LIN {X 0,Y 258.679,Z 819.95,A -85,B 0,C 180,E1 17212.36,E2 17212.36} C_VEL
LIN {X 0,Y 264.496,Z 801.8,A -85,B 0,C 180,E1 17220.057,E2 17220.057} C_VEL
LIN {X 0,Y 273.241,Z 778.314,A -85,B 0,C 180,E1 17227.008,E2 17227.008} C_VEL
LIN {X 0,Y 284.7,Z 748.46,A -85,B 0,C 180,E1 17233.215,E2 17233.215} C_VEL
LIN {X 0,Y 297.106,Z 713.594,A -85,B 0,C 180,E1 17238.218,E2 17238.218} C_VEL
LIN {X 0,Y 308.167,Z 677.358,A -85,B 0,C 180,E1 17241.821,E2 17241.821} C_VEL
LIN {X 0,Y 310.723,Z 665.135,A -85,B 0,C 180,E1 17242.87,E2 17242.87} C_VEL
LIN {X 0,Y 299.112,Z 634.221,A -85,B 0,C 180,E1 17248.073,E2 17248.073} C_VEL
LIN {X 0,Y 298.499,Z 632.776,A -85,B 0,C 180,E1 17248.333,E2 17248.333} C_VEL
LIN {X 0,Y 292.941,Z 625.387,A -85,B 0,C 180,E1 17250.142,E2 17250.142} C_VEL
LIN {X 0,Y 282.487,Z 614.328,A -85,B 0,C 180,E1 17253.334,E2 17253.334} C_VEL
LIN {X 0,Y 266.688,Z 585.354,A -85,B 0,C 180,E1 17259.767,E2 17259.767} C_VEL
LIN {X 0,Y 252.053,Z 561.723,A -85,B 0,C 180,E1 17266.216,E2 17266.216} C_VEL
LIN {X 0,Y 248.005,Z 555.389,A -85,B 0,C 180,E1 17268.238,E2 17268.238} C_VEL
LIN {X 0,Y 245.574,Z 550.181,A -85,B 0,C 180,E1 17269.651,E2 17269.651} C_VEL
LIN {X 0,Y 246.167,Z 549.53,A -85,B 0,C 180,E1 17276.481,E2 17276.481} C_VEL
LIN {X 0,Y 246.53,Z 549.53,A -85,B 0,C 180,E1 17280.007,E2 17280.007} C_VEL
LIN {X 0,Y 245.808,Z 549.53,A -85,B 0,C 180,E1 17287.084,E2 17287.084} C_VEL
LIN {X 0,Y 245.168,Z 549.53,A -85,B 0,C 180,E1 17294.309,E2 17294.309} C_VEL
LIN {X 0,Y 244.572,Z 549.53,A -85,B 0,C 180,E1 17301.812,E2 17301.812} C_VEL
LIN {X 0,Y 244.107,Z 549.53,A -85,B 0,C 180,E1 17309.756,E2 17309.756} C_VEL
LIN {X 0,Y 243.773,Z 549.53,A -85,B 0,C 180,E1 17318.404,E2 17318.404} C_VEL
LIN {X 0,Y 243.66,Z 549.53,A -85,B 0,C 180,E1 17326.882,E2 17326.882} C_VEL
LIN {X 0,Y 243.817,Z 549.53,A -85,B 0,C 180,E1 17336.023,E2 17336.023} C_VEL
LIN {X 0,Y 244.37,Z 549.53,A -85,B 0,C 180,E1 17344.299,E2 17344.299} C_VEL
LIN {X 0,Y 244.862,Z 549.53,A -85,B 0,C 180,E1 17351.993,E2 17351.993} C_VEL
LIN {X 0,Y 245.584,Z 549.53,A -85,B 0,C 180,E1 17360.585,E2 17360.585} C_VEL
LIN {X 0,Y 246.312,Z 549.696,A -85,B 0,C 180,E1 17368.13,E2 17368.13} C_VEL
LIN {X 0,Y 248.757,Z 555.053,A -85,B 0,C 180,E1 17369.566,E2 17369.566} C_VEL
LIN {X 0,Y 251.1,Z 558.751,A -85,B 0,C 180,E1 17370.757,E2 17370.757} C_VEL
LIN {X 0,Y 263.419,Z 580.328,A -85,B 0,C 180,E1 17376.986,E2 17376.986} C_VEL
LIN {X 0,Y 276.368,Z 608.507,A -85,B 0,C 180,E1 17383.801,E2 17383.801} C_VEL
LIN {X 0,Y 286.352,Z 636.818,A -85,B 0,C 180,E1 17389.901,E2 17389.901} C_VEL
LIN {X 0,Y 293.204,Z 665.582,A -85,B 0,C 180,E1 17395.869,E2 17395.869} C_VEL
LIN {X 0,Y 292.815,Z 670.961,A -85,B 0,C 180,E1 17396.759,E2 17396.759} C_VEL
LIN {X 0,Y 280.786,Z 703.835,A -85,B 0,C 180,E1 17401.766,E2 17401.766} C_VEL
LIN {X 0,Y 269.635,Z 731.204,A -85,B 0,C 180,E1 17407.633,E2 17407.633} C_VEL
LIN {X 0,Y 260.58,Z 753.078,A -85,B 0,C 180,E1 17414.208,E2 17414.208} C_VEL
LIN {X 0,Y 253.504,Z 771.169,A -85,B 0,C 180,E1 17421.942,E2 17421.942} C_VEL
LIN {X 0,Y 249.653,Z 783.095,A -85,B 0,C 180,E1 17429.414,E2 17429.414} C_VEL
LIN {X 0,Y 247.652,Z 790.352,A -85,B 0,C 180,E1 17436.502,E2 17436.502} C_VEL
LIN {X 0,Y 246.858,Z 793.707,A -85,B 0,C 180,E1 17442.134,E2 17442.134} C_VEL
LIN {X 0,Y 247.311,Z 795.056,A -85,B 0,C 180,E1 17449.41,E2 17449.41} C_VEL
LIN {X 0,Y 249.686,Z 792.262,A -85,B 0,C 180,E1 17458.054,E2 17458.054} C_VEL
LIN {X 0,Y 255.266,Z 783.653,A -85,B 0,C 180,E1 17467.662,E2 17467.662} C_VEL
LIN {X 0,Y 265.509,Z 769.339,A -85,B 0,C 180,E1 17476.559,E2 17476.559} C_VEL
LIN {X 0,Y 280.933,Z 748.975,A -85,B 0,C 180,E1 17484.68,E2 17484.68} C_VEL
LIN {X 0,Y 304.019,Z 719.389,A -85,B 0,C 180,E1 17492.361,E2 17492.361} C_VEL
LIN {X 0,Y 315.827,Z 704.851,A -85,B 0,C 180,E1 17495.111,E2 17495.111} C_VEL
LIN {X 0,Y 317.542,Z 702.998,A -85,B 0,C 180,E1 17495.846,E2 17495.846} C_VEL
LIN {X 0,Y 291.865,Z 741.185,A -85,B 0,C 180,E1 17501.778,E2 17501.778} C_VEL
LIN {X 0,Y 271.633,Z 776.074,A -85,B 0,C 180,E1 17509.609,E2 17509.609} C_VEL
LIN {X 0,Y 258.491,Z 802.354,A -85,B 0,C 180,E1 17518.185,E2 17518.185} C_VEL
LIN {X 0,Y 251.091,Z 820.776,A -85,B 0,C 180,E1 17526.923,E2 17526.923} C_VEL
LIN {X 0,Y 247.867,Z 833.059,A -85,B 0,C 180,E1 17535.856,E2 17535.856} C_VEL
LIN {X 0,Y 247.295,Z 838.614,A -85,B 0,C 180,E1 17542.965,E2 17542.965} C_VEL
LIN {X 0,Y 247.721,Z 840.447,A -85,B 0,C 180,E1 17549.998,E2 17549.998} C_VEL
LIN {X 0,Y 247.391,Z 838.37,A -85,B 0,C 180,E1 17557.029,E2 17557.029} C_VEL
LIN {X 0,Y 248.174,Z 831.193,A -85,B 0,C 180,E1 17565.026,E2 17565.026} C_VEL
LIN {X 0,Y 251.104,Z 818.708,A -85,B 0,C 180,E1 17573.073,E2 17573.073} C_VEL
LIN {X 0,Y 257.828,Z 799.096,A -85,B 0,C 180,E1 17581.409,E2 17581.409} C_VEL
LIN {X 0,Y 267.398,Z 774.73,A -85,B 0,C 180,E1 17588.522,E2 17588.522} C_VEL
LIN {X 0,Y 279.477,Z 743.888,A -85,B 0,C 180,E1 17594.769,E2 17594.769} C_VEL
LIN {X 0,Y 291.672,Z 710.486,A -85,B 0,C 180,E1 17599.468,E2 17599.468} C_VEL
LIN {X 0,Y 303.095,Z 673.739,A -85,B 0,C 180,E1 17603.057,E2 17603.057} C_VEL
LIN {X 0,Y 304.159,Z 667.908,A -85,B 0,C 180,E1 17603.602,E2 17603.602} C_VEL
LIN {X 0,Y 292.207,Z 635.748,A -85,B 0,C 180,E1 17609.233,E2 17609.233} C_VEL
LIN {X 0,Y 282.487,Z 614.328,A -85,B 0,C 180,E1 17613.334,E2 17613.334} C_VEL
LIN {X 0,Y 276.396,Z 609.661,A -85,B 0,C 180,E1 17615.17,E2 17615.17} C_VEL
LIN {X 0,Y 270.283,Z 605.228,A -85,B 0,C 180,E1 17617.101,E2 17617.101} C_VEL
LIN {X 0,Y 254.507,Z 577.634,A -85,B 0,C 180,E1 17624.093,E2 17624.093} C_VEL
LIN {X 0,Y 244.101,Z 561.372,A -85,B 0,C 180,E1 17629.196,E2 17629.196} C_VEL
LIN {X 0,Y 240.425,Z 555.492,A -85,B 0,C 180,E1 17631.212,E2 17631.212} C_VEL
LIN {X 0,Y 237.922,Z 550.392,A -85,B 0,C 180,E1 17632.811,E2 17632.811} C_VEL
LIN {X 0,Y 237.963,Z 549.53,A -85,B 0,C 180,E1 17634.531,E2 17634.531} C_VEL
LIN {X 0,Y 238.619,Z 549.53,A -85,B 0,C 180,E1 17640.008,E2 17640.008} C_VEL
LIN {X 0,Y 237.871,Z 549.53,A -85,B 0,C 180,E1 17647.321,E2 17647.321} C_VEL
LIN {X 0,Y 236.963,Z 549.53,A -85,B 0,C 180,E1 17656.586,E2 17656.586} C_VEL
LIN {X 0,Y 236.356,Z 549.53,A -85,B 0,C 180,E1 17666.26,E2 17666.26} C_VEL
LIN {X 0,Y 235.845,Z 549.53,A -85,B 0,C 180,E1 17675.303,E2 17675.303} C_VEL
LIN {X 0,Y 235.738,Z 549.53,A -85,B 0,C 180,E1 17679.97,E2 17679.97} C_VEL
LIN {X 0,Y 235.649,Z 549.53,A -85,B 0,C 180,E1 17685.03,E2 17685.03} C_VEL
LIN {X 0,Y 235.739,Z 549.53,A -85,B 0,C 180,E1 17690.429,E2 17690.429} C_VEL
LIN {X 0,Y 236.003,Z 549.53,A -85,B 0,C 180,E1 17699.122,E2 17699.122} C_VEL
LIN {X 0,Y 236.549,Z 549.53,A -85,B 0,C 180,E1 17707.418,E2 17707.418} C_VEL
LIN {X 0,Y 237.187,Z 549.53,A -85,B 0,C 180,E1 17715.208,E2 17715.208} C_VEL
LIN {X 0,Y 238.025,Z 549.53,A -85,B 0,C 180,E1 17724.641,E2 17724.641} C_VEL
LIN {X 0,Y 240.769,Z 555.222,A -85,B 0,C 180,E1 17726.498,E2 17726.498} C_VEL
LIN {X 0,Y 243.309,Z 558.602,A -85,B 0,C 180,E1 17727.84,E2 17727.84} C_VEL
LIN {X 0,Y 250.787,Z 570.99,A -85,B 0,C 180,E1 17731.948,E2 17731.948} C_VEL
LIN {X 0,Y 263.707,Z 596.414,A -85,B 0,C 180,E1 17739.024,E2 17739.024} C_VEL
LIN {X 0,Y 274.879,Z 623.995,A -85,B 0,C 180,E1 17745.578,E2 17745.578} C_VEL
LIN {X 0,Y 282.972,Z 651.486,A -85,B 0,C 180,E1 17751.585,E2 17751.585} C_VEL
LIN {X 0,Y 286.801,Z 670.97,A -85,B 0,C 180,E1 17755.735,E2 17755.735} C_VEL
LIN {X 0,Y 274.284,Z 704.137,A -85,B 0,C 180,E1 17760.819,E2 17760.819} C_VEL
LIN {X 0,Y 262.588,Z 731.978,A -85,B 0,C 180,E1 17766.891,E2 17766.891} C_VEL
LIN {X 0,Y 252.725,Z 754.95,A -85,B 0,C 180,E1 17774.026,E2 17774.026} C_VEL
LIN {X 0,Y 245.589,Z 772.629,A -85,B 0,C 180,E1 17781.931,E2 17781.931} C_VEL
LIN {X 0,Y 241.565,Z 784.643,A -85,B 0,C 180,E1 17789.898,E2 17789.898} C_VEL
LIN {X 0,Y 239.57,Z 792.041,A -85,B 0,C 180,E1 17797.709,E2 17797.709} C_VEL
LIN {X 0,Y 238.952,Z 795.448,A -85,B 0,C 180,E1 17805.311,E2 17805.311} C_VEL
LIN {X 0,Y 240.119,Z 795.517,A -85,B 0,C 180,E1 17812.748,E2 17812.748} C_VEL
LIN {X 0,Y 243.453,Z 791.274,A -85,B 0,C 180,E1 17821.774,E2 17821.774} C_VEL
LIN {X 0,Y 250.937,Z 781.385,A -85,B 0,C 180,E1 17831.301,E2 17831.301} C_VEL
LIN {X 0,Y 263.563,Z 765.709,A -85,B 0,C 180,E1 17840.154,E2 17840.154} C_VEL
LIN {X 0,Y 282.697,Z 743.043,A -85,B 0,C 180,E1 17848.372,E2 17848.372} C_VEL
LIN {X 0,Y 308.114,Z 714.215,A -85,B 0,C 180,E1 17855.258,E2 17855.258} C_VEL
LIN {X 0,Y 308.844,Z 713.437,A -85,B 0,C 180,E1 17855.408,E2 17855.408} C_VEL
LIN {X 0,Y 302.639,Z 721.468,A -85,B 0,C 180,E1 17856.824,E2 17856.824} C_VEL
LIN {X 0,Y 277.298,Z 757.741,A -85,B 0,C 180,E1 17863.687,E2 17863.687} C_VEL
LIN {X 0,Y 259.124,Z 788.04,A -85,B 0,C 180,E1 17872.013,E2 17872.013} C_VEL
LIN {X 0,Y 247.804,Z 810.105,A -85,B 0,C 180,E1 17880.737,E2 17880.737} C_VEL
LIN {X 0,Y 241.66,Z 825.984,A -85,B 0,C 180,E1 17889.99,E2 17889.99} C_VEL
LIN {X 0,Y 239.571,Z 835.597,A -85,B 0,C 180,E1 17899.069,E2 17899.069} C_VEL
LIN {X 0,Y 239.542,Z 839.221,A -85,B 0,C 180,E1 17906.375,E2 17906.375} C_VEL
LIN {X 0,Y 239.852,Z 839.639,A -85,B 0,C 180,E1 17909.998,E2 17909.998} C_VEL
LIN {X 0,Y 239.513,Z 837.435,A -85,B 0,C 180,E1 17917.262,E2 17917.262} C_VEL
LIN {X 0,Y 240.411,Z 830.134,A -85,B 0,C 180,E1 17925.523,E2 17925.523} C_VEL
LIN {X 0,Y 243.569,Z 817.425,A -85,B 0,C 180,E1 17933.83,E2 17933.83} C_VEL
LIN {X 0,Y 250.598,Z 797.946,A -85,B 0,C 180,E1 17942.253,E2 17942.253} C_VEL
LIN {X 0,Y 260.897,Z 772.762,A -85,B 0,C 180,E1 17949.668,E2 17949.668} C_VEL
LIN {X 0,Y 273.176,Z 742.586,A -85,B 0,C 180,E1 17955.81,E2 17955.81} C_VEL
LIN {X 0,Y 285.963,Z 708.385,A -85,B 0,C 180,E1 17960.629,E2 17960.629} C_VEL
LIN {X 0,Y 297.463,Z 670.312,A -85,B 0,C 180,E1 17964.393,E2 17964.393} C_VEL
LIN {X 0,Y 286.549,Z 640.248,A -85,B 0,C 180,E1 17969.878,E2 17969.878} C_VEL
LIN {X 0,Y 272.704,Z 609.927,A -85,B 0,C 180,E1 17976.055,E2 17976.055} C_VEL
LIN {X 0,Y 270.283,Z 605.228,A -85,B 0,C 180,E1 17977.101,E2 17977.101} C_VEL
LIN {X 0,Y 264.394,Z 600.927,A -85,B 0,C 180,E1 17979.078,E2 17979.078} C_VEL
LIN {X 0,Y 258.27,Z 597.088,A -85,B 0,C 180,E1 17981.165,E2 17981.165} C_VEL
LIN {X 0,Y 244.464,Z 573.7,A -85,B 0,C 180,E1 17987.943,E2 17987.943} C_VEL
LIN {X 0,Y 236.484,Z 561.386,A -85,B 0,C 180,E1 17992.304,E2 17992.304} C_VEL
LIN {X 0,Y 233.266,Z 555.895,A -85,B 0,C 180,E1 17994.304,E2 17994.304} C_VEL
LIN {X 0,Y 230.424,Z 550.718,A -85,B 0,C 180,E1 17996.241,E2 17996.241} C_VEL
LIN {X 0,Y 230.341,Z 549.53,A -85,B 0,C 180,E1 17996.711,E2 17996.711} C_VEL
LIN {X 0,Y 230.707,Z 549.53,A -85,B 0,C 180,E1 18000.008,E2 18000.008} C_VEL
LIN {X 0,Y 229.724,Z 549.53,A -85,B 0,C 180,E1 18008.663,E2 18008.663} C_VEL
LIN {X 0,Y 229.174,Z 549.53,A -85,B 0,C 180,E1 18015.331,E2 18015.331} C_VEL
LIN {X 0,Y 228.512,Z 549.53,A -85,B 0,C 180,E1 18023.433,E2 18023.433} C_VEL
LIN {X 0,Y 228.009,Z 549.53,A -85,B 0,C 180,E1 18032.097,E2 18032.097} C_VEL
LIN {X 0,Y 227.602,Z 549.53,A -85,B 0,C 180,E1 18041.709,E2 18041.709} C_VEL
LIN {X 0,Y 227.597,Z 549.53,A -85,B 0,C 180,E1 18048.302,E2 18048.302} C_VEL
LIN {X 0,Y 228.009,Z 549.53,A -85,B 0,C 180,E1 18057.913,E2 18057.913} C_VEL
LIN {X 0,Y 228.645,Z 549.53,A -85,B 0,C 180,E1 18068,E2 18068} C_VEL
LIN {X 0,Y 229.199,Z 549.53,A -85,B 0,C 180,E1 18074.68,E2 18074.68} C_VEL
LIN {X 0,Y 229.754,Z 550.148,A -85,B 0,C 180,E1 18081.018,E2 18081.018} C_VEL
LIN {X 0,Y 232.751,Z 555.489,A -85,B 0,C 180,E1 18083.054,E2 18083.054} C_VEL
LIN {X 0,Y 234.928,Z 558.032,A -85,B 0,C 180,E1 18084.338,E2 18084.338} C_VEL
LIN {X 0,Y 243.185,Z 570.639,A -85,B 0,C 180,E1 18089.204,E2 18089.204} C_VEL
LIN {X 0,Y 254.741,Z 593.004,A -85,B 0,C 180,E1 18095.972,E2 18095.972} C_VEL
LIN {X 0,Y 265.643,Z 618.495,A -85,B 0,C 180,E1 18102.565,E2 18102.565} C_VEL
LIN {X 0,Y 274.339,Z 645.864,A -85,B 0,C 180,E1 18108.921,E2 18108.921} C_VEL
LIN {X 0,Y 279.945,Z 672.119,A -85,B 0,C 180,E1 18114.758,E2 18114.758} C_VEL
LIN {X 0,Y 267.572,Z 705.02,A -85,B 0,C 180,E1 18119.97,E2 18119.97} C_VEL
LIN {X 0,Y 255.483,Z 732.854,A -85,B 0,C 180,E1 18126.158,E2 18126.158} C_VEL
LIN {X 0,Y 245.566,Z 755.151,A -85,B 0,C 180,E1 18133.211,E2 18133.211} C_VEL
LIN {X 0,Y 237.953,Z 773.25,A -85,B 0,C 180,E1 18141.461,E2 18141.461} C_VEL
LIN {X 0,Y 233.463,Z 786.339,A -85,B 0,C 180,E1 18150.561,E2 18150.561} C_VEL
LIN {X 0,Y 231.456,Z 793.487,A -85,B 0,C 180,E1 18158.905,E2 18158.905} C_VEL
LIN {X 0,Y 231.427,Z 796.695,A -85,B 0,C 180,E1 18168.673,E2 18168.673} C_VEL
LIN {X 0,Y 233.244,Z 795.585,A -85,B 0,C 180,E1 18176.27,E2 18176.27} C_VEL
LIN {X 0,Y 237.874,Z 790.072,A -85,B 0,C 180,E1 18185.471,E2 18185.471} C_VEL
LIN {X 0,Y 247.546,Z 778.881,A -85,B 0,C 180,E1 18195.059,E2 18195.059} C_VEL
LIN {X 0,Y 264.487,Z 760.213,A -85,B 0,C 180,E1 18204.513,E2 18204.513} C_VEL
LIN {X 0,Y 290.478,Z 732.854,A -85,B 0,C 180,E1 18213.16,E2 18213.16} C_VEL
LIN {X 0,Y 299.683,Z 723.675,A -85,B 0,C 180,E1 18215.291,E2 18215.291} C_VEL
LIN {X 0,Y 267.055,Z 766.39,A -85,B 0,C 180,E1 18224.291,E2 18224.291} C_VEL
LIN {X 0,Y 248.352,Z 795.614,A -85,B 0,C 180,E1 18233.528,E2 18233.528} C_VEL
LIN {X 0,Y 237.716,Z 815.993,A -85,B 0,C 180,E1 18243.067,E2 18243.067} C_VEL
LIN {X 0,Y 232.727,Z 829.792,A -85,B 0,C 180,E1 18252.975,E2 18252.975} C_VEL
LIN {X 0,Y 231.605,Z 836.164,A -85,B 0,C 180,E1 18260.592,E2 18260.592} C_VEL
LIN {X 0,Y 231.671,Z 838.445,A -85,B 0,C 180,E1 18266.251,E2 18266.251} C_VEL
LIN {X 0,Y 231.996,Z 838.833,A -85,B 0,C 180,E1 18269.998,E2 18269.998} C_VEL
LIN {X 0,Y 231.656,Z 836.479,A -85,B 0,C 180,E1 18277.509,E2 18277.509} C_VEL
LIN {X 0,Y 232.635,Z 829.058,A -85,B 0,C 180,E1 18286.056,E2 18286.056} C_VEL
LIN {X 0,Y 236.082,Z 816.119,A -85,B 0,C 180,E1 18294.635,E2 18294.635} C_VEL
LIN {X 0,Y 243.376,Z 796.854,A -85,B 0,C 180,E1 18303.097,E2 18303.097} C_VEL
LIN {X 0,Y 253.891,Z 772.146,A -85,B 0,C 180,E1 18310.505,E2 18310.505} C_VEL
LIN {X 0,Y 266.467,Z 742.247,A -85,B 0,C 180,E1 18316.717,E2 18316.717} C_VEL
LIN {X 0,Y 279.353,Z 709.063,A -85,B 0,C 180,E1 18321.488,E2 18321.488} C_VEL
LIN {X 0,Y 290.888,Z 673.4,A -85,B 0,C 180,E1 18325.081,E2 18325.081} C_VEL
LIN {X 0,Y 280.177,Z 642.883,A -85,B 0,C 180,E1 18330.907,E2 18330.907} C_VEL
LIN {X 0,Y 266.829,Z 613.087,A -85,B 0,C 180,E1 18337.219,E2 18337.219} C_VEL
LIN {X 0,Y 258.27,Z 597.088,A -85,B 0,C 180,E1 18341.165,E2 18341.165} C_VEL
LIN {X 0,Y 252.244,Z 593.691,A -85,B 0,C 180,E1 18343.355,E2 18343.355} C_VEL
LIN {X 0,Y 247.193,Z 590.636,A -85,B 0,C 180,E1 18345.306,E2 18345.306} C_VEL
LIN {X 0,Y 246.713,Z 589.779,A -85,B 0,C 180,E1 18345.56,E2 18345.56} C_VEL
LIN {X 0,Y 234.069,Z 568.962,A -85,B 0,C 180,E1 18352.575,E2 18352.575} C_VEL
LIN {X 0,Y 226.044,Z 556.135,A -85,B 0,C 180,E1 18357.823,E2 18357.823} C_VEL
LIN {X 0,Y 222.931,Z 551.116,A -85,B 0,C 180,E1 18360.13,E2 18360.13} C_VEL
LIN {X 0,Y 222.697,Z 549.53,A -85,B 0,C 180,E1 18360.495,E2 18360.495} C_VEL
LIN {X 0,Y 221.947,Z 549.53,A -85,B 0,C 180,E1 18367.85,E2 18367.85} C_VEL
LIN {X 0,Y 221.048,Z 549.53,A -85,B 0,C 180,E1 18376.484,E2 18376.484} C_VEL
LIN {X 0,Y 220.435,Z 549.53,A -85,B 0,C 180,E1 18384.346,E2 18384.346} C_VEL
LIN {X 0,Y 219.882,Z 549.53,A -85,B 0,C 180,E1 18393.435,E2 18393.435} C_VEL
LIN {X 0,Y 219.643,Z 549.53,A -85,B 0,C 180,E1 18403.587,E2 18403.587} C_VEL
LIN {X 0,Y 219.657,Z 549.53,A -85,B 0,C 180,E1 18411.66,E2 18411.66} C_VEL
LIN {X 0,Y 220.217,Z 549.53,A -85,B 0,C 180,E1 18421.233,E2 18421.233} C_VEL
LIN {X 0,Y 220.82,Z 549.53,A -85,B 0,C 180,E1 18429.953,E2 18429.953} C_VEL
LIN {X 0,Y 221.355,Z 550.069,A -85,B 0,C 180,E1 18436.529,E2 18436.529} C_VEL
LIN {X 0,Y 224.335,Z 555.453,A -85,B 0,C 180,E1 18438.897,E2 18438.897} C_VEL
LIN {X 0,Y 226.792,Z 558.2,A -85,B 0,C 180,E1 18440.56,E2 18440.56} C_VEL
LIN {X 0,Y 236.076,Z 571.606,A -85,B 0,C 180,E1 18446.543,E2 18446.543} C_VEL
LIN {X 0,Y 245.543,Z 589.276,A -85,B 0,C 180,E1 18452.513,E2 18452.513} C_VEL
LIN {X 0,Y 256.939,Z 614.863,A -85,B 0,C 180,E1 18459.755,E2 18459.755} C_VEL
LIN {X 0,Y 265.719,Z 640.684,A -85,B 0,C 180,E1 18466.129,E2 18466.129} C_VEL
LIN {X 0,Y 272.22,Z 668.713,A -85,B 0,C 180,E1 18472.661,E2 18472.661} C_VEL
LIN {X 0,Y 272.831,Z 676.317,A -85,B 0,C 180,E1 18474.308,E2 18474.308} C_VEL
LIN {X 0,Y 260.001,Z 708.083,A -85,B 0,C 180,E1 18479.504,E2 18479.504} C_VEL
LIN {X 0,Y 247.661,Z 735.405,A -85,B 0,C 180,E1 18485.853,E2 18485.853} C_VEL
LIN {X 0,Y 237.076,Z 758.304,A -85,B 0,C 180,E1 18493.512,E2 18493.512} C_VEL
LIN {X 0,Y 229.424,Z 776.284,A -85,B 0,C 180,E1 18502.369,E2 18502.369} C_VEL
LIN {X 0,Y 225.183,Z 788.683,A -85,B 0,C 180,E1 18511.915,E2 18511.915} C_VEL
LIN {X 0,Y 223.414,Z 794.916,A -85,B 0,C 180,E1 18520.185,E2 18520.185} C_VEL
LIN {X 0,Y 223.507,Z 797.499,A -85,B 0,C 180,E1 18528.266,E2 18528.266} C_VEL
LIN {X 0,Y 225.359,Z 796.753,A -85,B 0,C 180,E1 18536.14,E2 18536.14} C_VEL
LIN {X 0,Y 230.148,Z 791.804,A -85,B 0,C 180,E1 18545.655,E2 18545.655} C_VEL
LIN {X 0,Y 241.456,Z 780.142,A -85,B 0,C 180,E1 18556.382,E2 18556.382} C_VEL
LIN {X 0,Y 259.683,Z 762.048,A -85,B 0,C 180,E1 18565.922,E2 18565.922} C_VEL
LIN {X 0,Y 287.372,Z 735.924,A -85,B 0,C 180,E1 18574.483,E2 18574.483} C_VEL
LIN {X 0,Y 289.92,Z 733.651,A -85,B 0,C 180,E1 18575.053,E2 18575.053} C_VEL
LIN {X 0,Y 289.574,Z 734.175,A -85,B 0,C 180,E1 18575.517,E2 18575.517} C_VEL
LIN {X 0,Y 261.636,Z 767.698,A -85,B 0,C 180,E1 18583.061,E2 18583.061} C_VEL
LIN {X 0,Y 242.601,Z 794.723,A -85,B 0,C 180,E1 18591.952,E2 18591.952} C_VEL
LIN {X 0,Y 230.832,Z 814.779,A -85,B 0,C 180,E1 18601.604,E2 18601.604} C_VEL
LIN {X 0,Y 225.307,Z 828.176,A -85,B 0,C 180,E1 18611.384,E2 18611.384} C_VEL
LIN {X 0,Y 223.726,Z 835.525,A -85,B 0,C 180,E1 18620.353,E2 18620.353} C_VEL
LIN {X 0,Y 223.798,Z 837.676,A -85,B 0,C 180,E1 18626.119,E2 18626.119} C_VEL
LIN {X 0,Y 224.147,Z 838.023,A -85,B 0,C 180,E1 18629.998,E2 18629.998} C_VEL
LIN {X 0,Y 223.805,Z 835.506,A -85,B 0,C 180,E1 18637.774,E2 18637.774} C_VEL
LIN {X 0,Y 224.878,Z 827.897,A -85,B 0,C 180,E1 18646.626,E2 18646.626} C_VEL
LIN {X 0,Y 228.669,Z 814.757,A -85,B 0,C 180,E1 18655.49,E2 18655.49} C_VEL
LIN {X 0,Y 236.915,Z 794.138,A -85,B 0,C 180,E1 18664.536,E2 18664.536} C_VEL
LIN {X 0,Y 247.479,Z 770.249,A -85,B 0,C 180,E1 18671.705,E2 18671.705} C_VEL
LIN {X 0,Y 260.641,Z 740.12,A -85,B 0,C 180,E1 18677.973,E2 18677.973} C_VEL
LIN {X 0,Y 274.039,Z 706.266,A -85,B 0,C 180,E1 18682.818,E2 18682.818} C_VEL
LIN {X 0,Y 284.19,Z 675.873,A -85,B 0,C 180,E1 18685.905,E2 18685.905} C_VEL
LIN {X 0,Y 273.387,Z 644.657,A -85,B 0,C 180,E1 18692.105,E2 18692.105} C_VEL
LIN {X 0,Y 260.762,Z 615.906,A -85,B 0,C 180,E1 18698.535,E2 18698.535} C_VEL
LIN {X 0,Y 246.713,Z 589.779,A -85,B 0,C 180,E1 18705.56,E2 18705.56} C_VEL
LIN {X 0,Y 241.268,Z 584.454,A -85,B 0,C 180,E1 18708.08,E2 18708.08} C_VEL
LIN {X 0,Y 232.959,Z 578.991,A -85,B 0,C 180,E1 18711.963,E2 18711.963} C_VEL
LIN {X 0,Y 231.959,Z 577.127,A -85,B 0,C 180,E1 18712.587,E2 18712.587} C_VEL
LIN {X 0,Y 222.439,Z 562.508,A -85,B 0,C 180,E1 18718.911,E2 18718.911} C_VEL
LIN {X 0,Y 218.926,Z 556.53,A -85,B 0,C 180,E1 18721.742,E2 18721.742} C_VEL
LIN {X 0,Y 214.411,Z 551.326,A -85,B 0,C 180,E1 18725.393,E2 18725.393} C_VEL
LIN {X 0,Y 214.142,Z 549.53,A -85,B 0,C 180,E1 18726.008,E2 18726.008} C_VEL
LIN {X 0,Y 213.551,Z 549.53,A -85,B 0,C 180,E1 18732.289,E2 18732.289} C_VEL
LIN {X 0,Y 212.566,Z 549.53,A -85,B 0,C 180,E1 18742.191,E2 18742.191} C_VEL
LIN {X 0,Y 211.989,Z 549.53,A -85,B 0,C 180,E1 18751.015,E2 18751.015} C_VEL
LIN {X 0,Y 211.706,Z 549.53,A -85,B 0,C 180,E1 18760.075,E2 18760.075} C_VEL
LIN {X 0,Y 211.7,Z 549.53,A -85,B 0,C 180,E1 18769.936,E2 18769.936} C_VEL
LIN {X 0,Y 212.084,Z 549.53,A -85,B 0,C 180,E1 18780.02,E2 18780.02} C_VEL
LIN {X 0,Y 212.75,Z 549.53,A -85,B 0,C 180,E1 18789.157,E2 18789.157} C_VEL
LIN {X 0,Y 212.96,Z 550.331,A -85,B 0,C 180,E1 18791.209,E2 18791.209} C_VEL
LIN {X 0,Y 215.857,Z 555.371,A -85,B 0,C 180,E1 18793.969,E2 18793.969} C_VEL
LIN {X 0,Y 218.538,Z 558.107,A -85,B 0,C 180,E1 18796.07,E2 18796.07} C_VEL
LIN {X 0,Y 224.393,Z 566.642,A -85,B 0,C 180,E1 18800.551,E2 18800.551} C_VEL
LIN {X 0,Y 232.286,Z 578.041,A -85,B 0,C 180,E1 18805.893,E2 18805.893} C_VEL
LIN {X 0,Y 242.56,Z 598.059,A -85,B 0,C 180,E1 18812.776,E2 18812.776} C_VEL
LIN {X 0,Y 253.342,Z 624.581,A -85,B 0,C 180,E1 18820.33,E2 18820.33} C_VEL
LIN {X 0,Y 261.202,Z 650.446,A -85,B 0,C 180,E1 18826.849,E2 18826.849} C_VEL
LIN {X 0,Y 266.372,Z 676.947,A -85,B 0,C 180,E1 18833.226,E2 18833.226} C_VEL
LIN {X 0,Y 253.394,Z 708.799,A -85,B 0,C 180,E1 18838.557,E2 18838.557} C_VEL
LIN {X 0,Y 240.544,Z 736.32,A -85,B 0,C 180,E1 18845.078,E2 18845.078} C_VEL
LIN {X 0,Y 229.127,Z 760.248,A -85,B 0,C 180,E1 18853.365,E2 18853.365} C_VEL
LIN {X 0,Y 221.683,Z 777.145,A -85,B 0,C 180,E1 18862.061,E2 18862.061} C_VEL
LIN {X 0,Y 217.268,Z 789.523,A -85,B 0,C 180,E1 18871.932,E2 18871.932} C_VEL
LIN {X 0,Y 215.611,Z 795.189,A -85,B 0,C 180,E1 18879.436,E2 18879.436} C_VEL
LIN {X 0,Y 215.763,Z 798.383,A -85,B 0,C 180,E1 18889.249,E2 18889.249} C_VEL
LIN {X 0,Y 219.085,Z 796.663,A -85,B 0,C 180,E1 18899.992,E2 18899.992} C_VEL
LIN {X 0,Y 225.64,Z 790.585,A -85,B 0,C 180,E1 18909.649,E2 18909.649} C_VEL
LIN {X 0,Y 239.783,Z 777.644,A -85,B 0,C 180,E1 18920.313,E2 18920.313} C_VEL
LIN {X 0,Y 262.691,Z 757.489,A -85,B 0,C 180,E1 18930.013,E2 18930.013} C_VEL
LIN {X 0,Y 280.956,Z 742.176,A -85,B 0,C 180,E1 18935.018,E2 18935.018} C_VEL
LIN {X 0,Y 244.931,Z 783.305,A -85,B 0,C 180,E1 18946.208,E2 18946.208} C_VEL
LIN {X 0,Y 228.063,Z 807.297,A -85,B 0,C 180,E1 18956.48,E2 18956.48} C_VEL
LIN {X 0,Y 219.431,Z 823.03,A -85,B 0,C 180,E1 18966.623,E2 18966.623} C_VEL
LIN {X 0,Y 216.282,Z 832.175,A -85,B 0,C 180,E1 18975.816,E2 18975.816} C_VEL
LIN {X 0,Y 215.778,Z 835.669,A -85,B 0,C 180,E1 18981.931,E2 18981.931} C_VEL
LIN {X 0,Y 216.289,Z 837.195,A -85,B 0,C 180,E1 18989.998,E2 18989.998} C_VEL
LIN {X 0,Y 215.948,Z 834.516,A -85,B 0,C 180,E1 18998.059,E2 18998.059} C_VEL
LIN {X 0,Y 217.14,Z 826.699,A -85,B 0,C 180,E1 19007.236,E2 19007.236} C_VEL
LIN {X 0,Y 221.591,Z 812.524,A -85,B 0,C 180,E1 19016.818,E2 19016.818} C_VEL
LIN {X 0,Y 229.643,Z 793.424,A -85,B 0,C 180,E1 19025.316,E2 19025.316} C_VEL
LIN {X 0,Y 241.283,Z 768.012,A -85,B 0,C 180,E1 19033.03,E2 19033.03} C_VEL
LIN {X 0,Y 254.503,Z 738.712,A -85,B 0,C 180,E1 19039.136,E2 19039.136} C_VEL
LIN {X 0,Y 268.891,Z 703.242,A -85,B 0,C 180,E1 19044.191,E2 19044.191} C_VEL
LIN {X 0,Y 277.346,Z 679.326,A -85,B 0,C 180,E1 19046.624,E2 19046.624} C_VEL
LIN {X 0,Y 269.884,Z 655.033,A -85,B 0,C 180,E1 19051.528,E2 19051.528} C_VEL
LIN {X 0,Y 258.232,Z 626.28,A -85,B 0,C 180,E1 19058,E2 19058} C_VEL
LIN {X 0,Y 244.12,Z 598.297,A -85,B 0,C 180,E1 19065.529,E2 19065.529} C_VEL
LIN {X 0,Y 231.959,Z 577.127,A -85,B 0,C 180,E1 19072.587,E2 19072.587} C_VEL
LIN {X 0,Y 228.112,Z 572.712,A -85,B 0,C 180,E1 19074.842,E2 19074.842} C_VEL
LIN {X 0,Y 218.719,Z 568.259,A -85,B 0,C 180,E1 19080.234,E2 19080.234} C_VEL
LIN {X 0,Y 218.397,Z 567.789,A -85,B 0,C 180,E1 19080.487,E2 19080.487} C_VEL
LIN {X 0,Y 215.673,Z 563.459,A -85,B 0,C 180,E1 19082.701,E2 19082.701} C_VEL
LIN {X 0,Y 211.4,Z 557.199,A -85,B 0,C 180,E1 19086.555,E2 19086.555} C_VEL
LIN {X 0,Y 206.023,Z 551.95,A -85,B 0,C 180,E1 19091.803,E2 19091.803} C_VEL
LIN {X 0,Y 205.544,Z 549.53,A -85,B 0,C 180,E1 19092.776,E2 19092.776} C_VEL
LIN {X 0,Y 204.718,Z 549.53,A -85,B 0,C 180,E1 19101.712,E2 19101.712} C_VEL
LIN {X 0,Y 204.047,Z 549.53,A -85,B 0,C 180,E1 19111.302,E2 19111.302} C_VEL
LIN {X 0,Y 203.82,Z 549.53,A -85,B 0,C 180,E1 19116.471,E2 19116.471} C_VEL
LIN {X 0,Y 203.676,Z 549.53,A -85,B 0,C 180,E1 19122.003,E2 19122.003} C_VEL
LIN {X 0,Y 203.678,Z 549.53,A -85,B 0,C 180,E1 19128.03,E2 19128.03} C_VEL
LIN {X 0,Y 203.896,Z 549.53,A -85,B 0,C 180,E1 19134.782,E2 19134.782} C_VEL
LIN {X 0,Y 204.482,Z 550.333,A -85,B 0,C 180,E1 19144.246,E2 19144.246} C_VEL
LIN {X 0,Y 207.56,Z 555.603,A -85,B 0,C 180,E1 19148.105,E2 19148.105} C_VEL
LIN {X 0,Y 210.204,Z 557.75,A -85,B 0,C 180,E1 19150.534,E2 19150.534} C_VEL
LIN {X 0,Y 214.464,Z 563.558,A -85,B 0,C 180,E1 19154.403,E2 19154.403} C_VEL
LIN {X 0,Y 222.141,Z 574.934,A -85,B 0,C 180,E1 19160.679,E2 19160.679} C_VEL
LIN {X 0,Y 230.571,Z 588.034,A -85,B 0,C 180,E1 19166.706,E2 19166.706} C_VEL
LIN {X 0,Y 241.381,Z 611.987,A -85,B 0,C 180,E1 19174.621,E2 19174.621} C_VEL
LIN {X 0,Y 250.394,Z 637.352,A -85,B 0,C 180,E1 19181.777,E2 19181.777} C_VEL
LIN {X 0,Y 256.699,Z 662.229,A -85,B 0,C 180,E1 19188.129,E2 19188.129} C_VEL
LIN {X 0,Y 259.231,Z 680.878,A -85,B 0,C 180,E1 19192.679,E2 19192.679} C_VEL
LIN {X 0,Y 245.046,Z 713.281,A -85,B 0,C 180,E1 19198.32,E2 19198.32} C_VEL
LIN {X 0,Y 231.207,Z 741.763,A -85,B 0,C 180,E1 19205.65,E2 19205.65} C_VEL
LIN {X 0,Y 220.347,Z 763.602,A -85,B 0,C 180,E1 19213.917,E2 19213.917} C_VEL
LIN {X 0,Y 213.064,Z 779.873,A -85,B 0,C 180,E1 19223.045,E2 19223.045} C_VEL
LIN {X 0,Y 209.326,Z 790.446,A -85,B 0,C 180,E1 19232.055,E2 19232.055} C_VEL
LIN {X 0,Y 207.46,Z 797.023,A -85,B 0,C 180,E1 19241.584,E2 19241.584} C_VEL
LIN {X 0,Y 208.37,Z 799.359,A -85,B 0,C 180,E1 19251.635,E2 19251.635} C_VEL
LIN {X 0,Y 212.082,Z 797.353,A -85,B 0,C 180,E1 19261.814,E2 19261.814} C_VEL
LIN {X 0,Y 222.144,Z 789.21,A -85,B 0,C 180,E1 19273.792,E2 19273.792} C_VEL
LIN {X 0,Y 239.385,Z 775.24,A -85,B 0,C 180,E1 19284.266,E2 19284.266} C_VEL
LIN {X 0,Y 266.441,Z 754.187,A -85,B 0,C 180,E1 19293.617,E2 19293.617} C_VEL
LIN {X 0,Y 271.55,Z 750.41,A -85,B 0,C 180,E1 19294.89,E2 19294.89} C_VEL
LIN {X 0,Y 235.113,Z 789.257,A -85,B 0,C 180,E1 19306.823,E2 19306.823} C_VEL
LIN {X 0,Y 218.7,Z 811.18,A -85,B 0,C 180,E1 19317.55,E2 19317.55} C_VEL
LIN {X 0,Y 210.372,Z 826.048,A -85,B 0,C 180,E1 19328.907,E2 19328.907} C_VEL
LIN {X 0,Y 208.003,Z 833.794,A -85,B 0,C 180,E1 19339.022,E2 19339.022} C_VEL
LIN {X 0,Y 208.023,Z 836.133,A -85,B 0,C 180,E1 19345.824,E2 19345.824} C_VEL
LIN {X 0,Y 208.434,Z 836.315,A -85,B 0,C 180,E1 19349.998,E2 19349.998} C_VEL
LIN {X 0,Y 208.102,Z 833.509,A -85,B 0,C 180,E1 19358.365,E2 19358.365} C_VEL
LIN {X 0,Y 209.389,Z 825.564,A -85,B 0,C 180,E1 19367.792,E2 19367.792} C_VEL
LIN {X 0,Y 213.587,Z 812.728,A -85,B 0,C 180,E1 19376.858,E2 19376.858} C_VEL
LIN {X 0,Y 222.574,Z 792.318,A -85,B 0,C 180,E1 19386.261,E2 19386.261} C_VEL
LIN {X 0,Y 234.403,Z 767.462,A -85,B 0,C 180,E1 19393.975,E2 19393.975} C_VEL
LIN {X 0,Y 248.213,Z 737.857,A -85,B 0,C 180,E1 19400.253,E2 19400.253} C_VEL
LIN {X 0,Y 262.64,Z 703.382,A -85,B 0,C 180,E1 19405.231,E2 19405.231} C_VEL
LIN {X 0,Y 270.745,Z 680.685,A -85,B 0,C 180,E1 19407.631,E2 19407.631} C_VEL
LIN {X 0,Y 260.785,Z 650.322,A -85,B 0,C 180,E1 19414.196,E2 19414.196} C_VEL
LIN {X 0,Y 249.848,Z 624.346,A -85,B 0,C 180,E1 19420.539,E2 19420.539} C_VEL
LIN {X 0,Y 236.428,Z 597.745,A -85,B 0,C 180,E1 19428.349,E2 19428.349} C_VEL
LIN {X 0,Y 224.01,Z 576.333,A -85,B 0,C 180,E1 19436.375,E2 19436.375} C_VEL
LIN {X 0,Y 218.397,Z 567.789,A -85,B 0,C 180,E1 19440.487,E2 19440.487} C_VEL
LIN {X 0,Y 213.991,Z 564.529,A -85,B 0,C 180,E1 19443.626,E2 19443.626} C_VEL
LIN {X 0,Y 206.37,Z 562.92,A -85,B 0,C 180,E1 19449.319,E2 19449.319} C_VEL
LIN {X 0,Y 203.166,Z 557.585,A -85,B 0,C 180,E1 19453.18,E2 19453.18} C_VEL
LIN {X 0,Y 196.904,Z 551.362,A -85,B 0,C 180,E1 19462.282,E2 19462.282} C_VEL
LIN {X 0,Y 196.472,Z 549.53,A -85,B 0,C 180,E1 19463.874,E2 19463.874} C_VEL
LIN {X 0,Y 195.984,Z 549.53,A -85,B 0,C 180,E1 19472.747,E2 19472.747} C_VEL
LIN {X 0,Y 195.612,Z 549.53,A -85,B 0,C 180,E1 19479.287,E2 19479.287} C_VEL
LIN {X 0,Y 195.514,Z 549.53,A -85,B 0,C 180,E1 19485.819,E2 19485.819} C_VEL
LIN {X 0,Y 195.967,Z 550.262,A -85,B 0,C 180,E1 19493.657,E2 19493.657} C_VEL
LIN {X 0,Y 199.474,Z 556.003,A -85,B 0,C 180,E1 19500.44,E2 19500.44} C_VEL
LIN {X 0,Y 202.134,Z 557.972,A -85,B 0,C 180,E1 19503.795,E2 19503.795} C_VEL
LIN {X 0,Y 205.752,Z 563.394,A -85,B 0,C 180,E1 19508.227,E2 19508.227} C_VEL
LIN {X 0,Y 207.809,Z 565.8,A -85,B 0,C 180,E1 19510.283,E2 19510.283} C_VEL
LIN {X 0,Y 213.209,Z 573.536,A -85,B 0,C 180,E1 19515.463,E2 19515.463} C_VEL
LIN {X 0,Y 221.041,Z 584.986,A -85,B 0,C 180,E1 19521.878,E2 19521.878} C_VEL
LIN {X 0,Y 229.328,Z 600.345,A -85,B 0,C 180,E1 19528.278,E2 19528.278} C_VEL
LIN {X 0,Y 238.976,Z 624.203,A -85,B 0,C 180,E1 19536.022,E2 19536.022} C_VEL
LIN {X 0,Y 246.46,Z 648.424,A -85,B 0,C 180,E1 19542.869,E2 19542.869} C_VEL
LIN {X 0,Y 251.723,Z 673.695,A -85,B 0,C 180,E1 19549.477,E2 19549.477} C_VEL
LIN {X 0,Y 252.322,Z 683.518,A -85,B 0,C 180,E1 19551.862,E2 19551.862} C_VEL
LIN {X 0,Y 237.435,Z 716.167,A -85,B 0,C 180,E1 19557.793,E2 19557.793} C_VEL
LIN {X 0,Y 223.928,Z 742.923,A -85,B 0,C 180,E1 19564.924,E2 19564.924} C_VEL
LIN {X 0,Y 213.211,Z 763.706,A -85,B 0,C 180,E1 19572.974,E2 19572.974} C_VEL
LIN {X 0,Y 205.314,Z 780.598,A -85,B 0,C 180,E1 19582.682,E2 19582.682} C_VEL
LIN {X 0,Y 201.735,Z 790.304,A -85,B 0,C 180,E1 19591.019,E2 19591.019} C_VEL
LIN {X 0,Y 199.627,Z 797.273,A -85,B 0,C 180,E1 19600.834,E2 19600.834} C_VEL
LIN {X 0,Y 200.426,Z 800.177,A -85,B 0,C 180,E1 19611.301,E2 19611.301} C_VEL
LIN {X 0,Y 203.373,Z 799.34,A -85,B 0,C 180,E1 19619.991,E2 19619.991} C_VEL
LIN {X 0,Y 212.514,Z 792.999,A -85,B 0,C 180,E1 19632.332,E2 19632.332} C_VEL
LIN {X 0,Y 229.164,Z 780.985,A -85,B 0,C 180,E1 19643.345,E2 19643.345} C_VEL
LIN {X 0,Y 258.125,Z 760.696,A -85,B 0,C 180,E1 19653.766,E2 19653.766} C_VEL
LIN {X 0,Y 261.691,Z 758.325,A -85,B 0,C 180,E1 19654.679,E2 19654.679} C_VEL
LIN {X 0,Y 257.661,Z 762.032,A -85,B 0,C 180,E1 19655.978,E2 19655.978} C_VEL
LIN {X 0,Y 227.519,Z 792.115,A -85,B 0,C 180,E1 19666.334,E2 19666.334} C_VEL
LIN {X 0,Y 209.608,Z 814.239,A -85,B 0,C 180,E1 19678.418,E2 19678.418} C_VEL
LIN {X 0,Y 201.767,Z 827.935,A -85,B 0,C 180,E1 19690.718,E2 19690.718} C_VEL
LIN {X 0,Y 199.996,Z 834.238,A -85,B 0,C 180,E1 19701.289,E2 19701.289} C_VEL
LIN {X 0,Y 200.598,Z 835.42,A -85,B 0,C 180,E1 19709.998,E2 19709.998} C_VEL
LIN {X 0,Y 200.25,Z 832.482,A -85,B 0,C 180,E1 19718.696,E2 19718.696} C_VEL
LIN {X 0,Y 201.676,Z 824.398,A -85,B 0,C 180,E1 19728.412,E2 19728.412} C_VEL
LIN {X 0,Y 206.736,Z 810.068,A -85,B 0,C 180,E1 19738.519,E2 19738.519} C_VEL
LIN {X 0,Y 216.21,Z 789.835,A -85,B 0,C 180,E1 19747.786,E2 19747.786} C_VEL
LIN {X 0,Y 229.422,Z 763.403,A -85,B 0,C 180,E1 19755.862,E2 19755.862} C_VEL
LIN {X 0,Y 244.306,Z 732.008,A -85,B 0,C 180,E1 19762.268,E2 19762.268} C_VEL
LIN {X 0,Y 258.831,Z 697.351,A -85,B 0,C 180,E1 19767.011,E2 19767.011} C_VEL
LIN {X 0,Y 263.857,Z 682.315,A -85,B 0,C 180,E1 19768.669,E2 19768.669} C_VEL
LIN {X 0,Y 254.372,Z 652.726,A -85,B 0,C 180,E1 19775.385,E2 19775.385} C_VEL
LIN {X 0,Y 243.206,Z 625.812,A -85,B 0,C 180,E1 19782.341,E2 19782.341} C_VEL
LIN {X 0,Y 230.671,Z 600.528,A -85,B 0,C 180,E1 19790.208,E2 19790.208} C_VEL
LIN {X 0,Y 219.315,Z 580.892,A -85,B 0,C 180,E1 19798.129,E2 19798.129} C_VEL
LIN {X 0,Y 212.828,Z 570.558,A -85,B 0,C 180,E1 19803.408,E2 19803.408} C_VEL
LIN {X 0,Y 207.683,Z 563.752,A -85,B 0,C 180,E1 19808.129,E2 19808.129} C_VEL
LIN {X 0,Y 206.37,Z 562.92,A -85,B 0,C 180,E1 19809.319,E2 19809.319} C_VEL
LIN {X 0,Y 196.741,Z 562.106,A -85,B 0,C 180,E1 19819.012,E2 19819.012} C_VEL
LIN {X 0,Y 194.386,Z 557.155,A -85,B 0,C 180,E1 19824.147,E2 19824.147} C_VEL
LIN {X 0,Y 190.631,Z 555.665,A -85,B 0,C 180,E1 19837.42,E2 19837.42} C_VEL
LIN {X 0,Y 193.823,Z 557.353,A -85,B 0,C 180,E1 19852.818,E2 19852.818} C_VEL
LIN {X 0,Y 197.116,Z 563.348,A -85,B 0,C 180,E1 19859.775,E2 19859.775} C_VEL
LIN {X 0,Y 199.752,Z 565.711,A -85,B 0,C 180,E1 19863.374,E2 19863.374} C_VEL
LIN {X 0,Y 204.224,Z 571.38,A -85,B 0,C 180,E1 19868.818,E2 19868.818} C_VEL
LIN {X 0,Y 213.576,Z 585.46,A -85,B 0,C 180,E1 19878.051,E2 19878.051} C_VEL
LIN {X 0,Y 222.696,Z 601.153,A -85,B 0,C 180,E1 19885.615,E2 19885.615} C_VEL
LIN {X 0,Y 231.946,Z 624.387,A -85,B 0,C 180,E1 19893.744,E2 19893.744} C_VEL
LIN {X 0,Y 239.432,Z 648.366,A -85,B 0,C 180,E1 19900.937,E2 19900.937} C_VEL
LIN {X 0,Y 244.517,Z 672.548,A -85,B 0,C 180,E1 19907.571,E2 19907.571} C_VEL
LIN {X 0,Y 245.654,Z 685.413,A -85,B 0,C 180,E1 19910.913,E2 19910.913} C_VEL
LIN {X 0,Y 230.789,Z 716.928,A -85,B 0,C 180,E1 19916.765,E2 19916.765} C_VEL
LIN {X 0,Y 216.479,Z 744.348,A -85,B 0,C 180,E1 19924.268,E2 19924.268} C_VEL
LIN {X 0,Y 205.501,Z 764.903,A -85,B 0,C 180,E1 19932.532,E2 19932.532} C_VEL
LIN {X 0,Y 197.626,Z 781.153,A -85,B 0,C 180,E1 19942.19,E2 19942.19} C_VEL
LIN {X 0,Y 193.511,Z 791.959,A -85,B 0,C 180,E1 19951.991,E2 19951.991} C_VEL
LIN {X 0,Y 191.705,Z 798.283,A -85,B 0,C 180,E1 19961.574,E2 19961.574} C_VEL
LIN {X 0,Y 192.45,Z 800.994,A -85,B 0,C 180,E1 19970.938,E2 19970.938} C_VEL
LIN {X 0,Y 195.479,Z 800.568,A -85,B 0,C 180,E1 19979.991,E2 19979.991} C_VEL
LIN {X 0,Y 205.032,Z 795.065,A -85,B 0,C 180,E1 19992.79,E2 19992.79} C_VEL
LIN {X 0,Y 224.186,Z 782.84,A -85,B 0,C 180,E1 20004.958,E2 20004.958} C_VEL
LIN {X 0,Y 252.124,Z 765.434,A -85,B 0,C 180,E1 20014.562,E2 20014.562} C_VEL
LIN {X 0,Y 234.345,Z 780.907,A -85,B 0,C 180,E1 20019.945,E2 20019.945} C_VEL
LIN {X 0,Y 209.207,Z 806.302,A -85,B 0,C 180,E1 20031.921,E2 20031.921} C_VEL
LIN {X 0,Y 196.449,Z 823.033,A -85,B 0,C 180,E1 20044.917,E2 20044.917} C_VEL
LIN {X 0,Y 192.478,Z 831.58,A -85,B 0,C 180,E1 20056.348,E2 20056.348} C_VEL
LIN {X 0,Y 192.26,Z 834.464,A -85,B 0,C 180,E1 20065.481,E2 20065.481} C_VEL
LIN {X 0,Y 192.756,Z 834.52,A -85,B 0,C 180,E1 20069.998,E2 20069.998} C_VEL
LIN {X 0,Y 192.392,Z 831.439,A -85,B 0,C 180,E1 20079.054,E2 20079.054} C_VEL
LIN {X 0,Y 193.74,Z 824.106,A -85,B 0,C 180,E1 20088.214,E2 20088.214} C_VEL
LIN {X 0,Y 198.685,Z 810.412,A -85,B 0,C 180,E1 20098.489,E2 20098.489} C_VEL
LIN {X 0,Y 208.323,Z 790.46,A -85,B 0,C 180,E1 20108.151,E2 20108.151} C_VEL
LIN {X 0,Y 221.191,Z 765.548,A -85,B 0,C 180,E1 20116.194,E2 20116.194} C_VEL
LIN {X 0,Y 236.183,Z 735.347,A -85,B 0,C 180,E1 20122.749,E2 20122.749} C_VEL
LIN {X 0,Y 251.83,Z 699.76,A -85,B 0,C 180,E1 20127.883,E2 20127.883} C_VEL
LIN {X 0,Y 257.219,Z 685.13,A -85,B 0,C 180,E1 20129.501,E2 20129.501} C_VEL
LIN {X 0,Y 247.935,Z 655.106,A -85,B 0,C 180,E1 20136.62,E2 20136.62} C_VEL
LIN {X 0,Y 237.173,Z 628.641,A -85,B 0,C 180,E1 20143.791,E2 20143.791} C_VEL
LIN {X 0,Y 225.239,Z 604.119,A -85,B 0,C 180,E1 20151.901,E2 20151.901} C_VEL
LIN {X 0,Y 214.042,Z 583.621,A -85,B 0,C 180,E1 20160.648,E2 20160.648} C_VEL
LIN {X 0,Y 209.442,Z 577.053,A -85,B 0,C 180,E1 20164.544,E2 20164.544} C_VEL
LIN {X 0,Y 204.976,Z 570.947,A -85,B 0,C 180,E1 20168.875,E2 20168.875} C_VEL
LIN {X 0,Y 200.876,Z 565.381,A -85,B 0,C 180,E1 20173.629,E2 20173.629} C_VEL
LIN {X 0,Y 196.741,Z 562.106,A -85,B 0,C 180,E1 20179.012,E2 20179.012} C_VEL
LIN {X 0,Y 193.184,Z 562.509,A -85,B 0,C 180,E1 20184.087,E2 20184.087} C_VEL
LIN {X 0,Y 190.328,Z 564.045,A -85,B 0,C 180,E1 20189.334,E2 20189.334} C_VEL
LIN {X 0,Y 188.825,Z 563.521,A -85,B 0,C 180,E1 20201.891,E2 20201.891} C_VEL
LIN {X 0,Y 191.806,Z 565.553,A -85,B 0,C 180,E1 20212.866,E2 20212.866} C_VEL
LIN {X 0,Y 195.771,Z 571.454,A -85,B 0,C 180,E1 20220.812,E2 20220.812} C_VEL
LIN {X 0,Y 197.354,Z 573.721,A -85,B 0,C 180,E1 20223.278,E2 20223.278} C_VEL
LIN {X 0,Y 203.083,Z 582.145,A -85,B 0,C 180,E1 20230.483,E2 20230.483} C_VEL
LIN {X 0,Y 206.626,Z 587.135,A -85,B 0,C 180,E1 20234.186,E2 20234.186} C_VEL
LIN {X 0,Y 216.157,Z 602.611,A -85,B 0,C 180,E1 20242.927,E2 20242.927} C_VEL
LIN {X 0,Y 223.737,Z 620.816,A -85,B 0,C 180,E1 20250.002,E2 20250.002} C_VEL
LIN {X 0,Y 231.691,Z 645.291,A -85,B 0,C 180,E1 20257.984,E2 20257.984} C_VEL
LIN {X 0,Y 236.92,Z 668.67,A -85,B 0,C 180,E1 20264.812,E2 20264.812} C_VEL
LIN {X 0,Y 239.222,Z 686.879,A -85,B 0,C 180,E1 20269.853,E2 20269.853} C_VEL
LIN {X 0,Y 223.814,Z 718.523,A -85,B 0,C 180,E1 20275.879,E2 20275.879} C_VEL
LIN {X 0,Y 209.269,Z 745.346,A -85,B 0,C 180,E1 20283.42,E2 20283.42} C_VEL
LIN {X 0,Y 197.346,Z 766.862,A -85,B 0,C 180,E1 20292.444,E2 20292.444} C_VEL
LIN {X 0,Y 189.09,Z 783.673,A -85,B 0,C 180,E1 20303.202,E2 20303.202} C_VEL
LIN {X 0,Y 185.007,Z 794.439,A -85,B 0,C 180,E1 20314.192,E2 20314.192} C_VEL
LIN {X 0,Y 183.815,Z 800.523,A -85,B 0,C 180,E1 20325.684,E2 20325.684} C_VEL
LIN {X 0,Y 185.716,Z 802.145,A -85,B 0,C 180,E1 20335.314,E2 20335.314} C_VEL
LIN {X 0,Y 190.036,Z 800.818,A -85,B 0,C 180,E1 20344.56,E2 20344.56} C_VEL
LIN {X 0,Y 202.611,Z 794.214,A -85,B 0,C 180,E1 20357.382,E2 20357.382} C_VEL
LIN {X 0,Y 226.641,Z 780.779,A -85,B 0,C 180,E1 20369.5,E2 20369.5} C_VEL
LIN {X 0,Y 241.816,Z 772.386,A -85,B 0,C 180,E1 20374.289,E2 20374.289} C_VEL
LIN {X 0,Y 240.793,Z 773.43,A -85,B 0,C 180,E1 20375.17,E2 20375.17} C_VEL
LIN {X 0,Y 210.388,Z 799.203,A -85,B 0,C 180,E1 20386.178,E2 20386.178} C_VEL
LIN {X 0,Y 192.839,Z 817.566,A -85,B 0,C 180,E1 20398.826,E2 20398.826} C_VEL
LIN {X 0,Y 185.761,Z 828.227,A -85,B 0,C 180,E1 20410.97,E2 20410.97} C_VEL
LIN {X 0,Y 184.259,Z 832.696,A -85,B 0,C 180,E1 20420.539,E2 20420.539} C_VEL
LIN {X 0,Y 184.916,Z 833.611,A -85,B 0,C 180,E1 20429.998,E2 20429.998} C_VEL
LIN {X 0,Y 184.598,Z 829.88,A -85,B 0,C 180,E1 20440.251,E2 20440.251} C_VEL
LIN {X 0,Y 186.515,Z 821.253,A -85,B 0,C 180,E1 20450.474,E2 20450.474} C_VEL
LIN {X 0,Y 192.695,Z 806.291,A -85,B 0,C 180,E1 20461.155,E2 20461.155} C_VEL
LIN {X 0,Y 204.06,Z 784.362,A -85,B 0,C 180,E1 20471.183,E2 20471.183} C_VEL
LIN {X 0,Y 217.997,Z 758.285,A -85,B 0,C 180,E1 20479.018,E2 20479.018} C_VEL
LIN {X 0,Y 233.945,Z 726.615,A -85,B 0,C 180,E1 20485.33,E2 20485.33} C_VEL
LIN {X 0,Y 249.665,Z 690.513,A -85,B 0,C 180,E1 20490.095,E2 20490.095} C_VEL
LIN {X 0,Y 250.369,Z 687.073,A -85,B 0,C 180,E1 20490.581,E2 20490.581} C_VEL
LIN {X 0,Y 241.44,Z 657.425,A -85,B 0,C 180,E1 20497.907,E2 20497.907} C_VEL
LIN {X 0,Y 230.992,Z 631.092,A -85,B 0,C 180,E1 20505.469,E2 20505.469} C_VEL
LIN {X 0,Y 219.865,Z 607.453,A -85,B 0,C 180,E1 20513.719,E2 20513.719} C_VEL
LIN {X 0,Y 210.004,Z 589.325,A -85,B 0,C 180,E1 20521.968,E2 20521.968} C_VEL
LIN {X 0,Y 205.32,Z 582.436,A -85,B 0,C 180,E1 20526.376,E2 20526.376} C_VEL
LIN {X 0,Y 202.152,Z 578.053,A -85,B 0,C 180,E1 20529.709,E2 20529.709} C_VEL
LIN {X 0,Y 197.505,Z 571.69,A -85,B 0,C 180,E1 20535.502,E2 20535.502} C_VEL
LIN {X 0,Y 192.613,Z 565.741,A -85,B 0,C 180,E1 20543.722,E2 20543.722} C_VEL
LIN {X 0,Y 190.328,Z 564.045,A -85,B 0,C 180,E1 20549.334,E2 20549.334} C_VEL
LIN {X 0,Y 188.717,Z 566.038,A -85,B 0,C 180,E1 20553.232,E2 20553.232} C_VEL
LIN {X 0,Y 186.822,Z 570.975,A -85,B 0,C 180,E1 20559.092,E2 20559.092} C_VEL
LIN {X 0,Y 186.768,Z 571.064,A -85,B 0,C 180,E1 20559.768,E2 20559.768} C_VEL
LIN {X 0,Y 189.612,Z 573.18,A -85,B 0,C 180,E1 20572.598,E2 20572.598} C_VEL
LIN {X 0,Y 193.793,Z 579.158,A -85,B 0,C 180,E1 20581.108,E2 20581.108} C_VEL
LIN {X 0,Y 200.224,Z 589.493,A -85,B 0,C 180,E1 20590.214,E2 20590.214} C_VEL
LIN {X 0,Y 205.934,Z 598.05,A -85,B 0,C 180,E1 20596.313,E2 20596.313} C_VEL
LIN {X 0,Y 213.704,Z 612.546,A -85,B 0,C 180,E1 20603.899,E2 20603.899} C_VEL
LIN {X 0,Y 221.428,Z 633.957,A -85,B 0,C 180,E1 20611.961,E2 20611.961} C_VEL
LIN {X 0,Y 227.762,Z 657.402,A -85,B 0,C 180,E1 20619.568,E2 20619.568} C_VEL
LIN {X 0,Y 231.681,Z 680.253,A -85,B 0,C 180,E1 20626.359,E2 20626.359} C_VEL
LIN {X 0,Y 232.611,Z 688.603,A -85,B 0,C 180,E1 20628.795,E2 20628.795} C_VEL
LIN {X 0,Y 216.983,Z 719.756,A -85,B 0,C 180,E1 20634.874,E2 20634.874} C_VEL
LIN {X 0,Y 202.209,Z 746.099,A -85,B 0,C 180,E1 20642.468,E2 20642.468} C_VEL
LIN {X 0,Y 189.438,Z 768.385,A -85,B 0,C 180,E1 20652.165,E2 20652.165} C_VEL
LIN {X 0,Y 181.339,Z 784.307,A -85,B 0,C 180,E1 20662.799,E2 20662.799} C_VEL
LIN {X 0,Y 177.398,Z 794.206,A -85,B 0,C 180,E1 20672.998,E2 20672.998} C_VEL
LIN {X 0,Y 175.881,Z 800.923,A -85,B 0,C 180,E1 20685.023,E2 20685.023} C_VEL
LIN {X 0,Y 177.733,Z 803.005,A -85,B 0,C 180,E1 20695.103,E2 20695.103} C_VEL
LIN {X 0,Y 182.369,Z 802.219,A -85,B 0,C 180,E1 20704.93,E2 20704.93} C_VEL
LIN {X 0,Y 195.363,Z 796.478,A -85,B 0,C 180,E1 20718.049,E2 20718.049} C_VEL
LIN {X 0,Y 220.341,Z 784.219,A -85,B 0,C 180,E1 20730.431,E2 20730.431} C_VEL
LIN {X 0,Y 232.303,Z 778.299,A -85,B 0,C 180,E1 20734.248,E2 20734.248} C_VEL
LIN {X 0,Y 231.215,Z 779.316,A -85,B 0,C 180,E1 20735.058,E2 20735.058} C_VEL
LIN {X 0,Y 199.911,Z 803.916,A -85,B 0,C 180,E1 20747.026,E2 20747.026} C_VEL
LIN {X 0,Y 183.488,Z 820.202,A -85,B 0,C 180,E1 20760.322,E2 20760.322} C_VEL
LIN {X 0,Y 177.383,Z 829.029,A -85,B 0,C 180,E1 20772.616,E2 20772.616} C_VEL
LIN {X 0,Y 176.37,Z 831.921,A -85,B 0,C 180,E1 20780.112,E2 20780.112} C_VEL
LIN {X 0,Y 177.048,Z 832.689,A -85,B 0,C 180,E1 20789.998,E2 20789.998} C_VEL
LIN {X 0,Y 176.735,Z 829.239,A -85,B 0,C 180,E1 20799.863,E2 20799.863} C_VEL
LIN {X 0,Y 178.423,Z 821.398,A -85,B 0,C 180,E1 20809.84,E2 20809.84} C_VEL
LIN {X 0,Y 184.237,Z 807.249,A -85,B 0,C 180,E1 20820.799,E2 20820.799} C_VEL
LIN {X 0,Y 194.765,Z 787.625,A -85,B 0,C 180,E1 20830.619,E2 20830.619} C_VEL
LIN {X 0,Y 209.047,Z 762.127,A -85,B 0,C 180,E1 20839.023,E2 20839.023} C_VEL
LIN {X 0,Y 226.051,Z 729.689,A -85,B 0,C 180,E1 20845.979,E2 20845.979} C_VEL
LIN {X 0,Y 242.113,Z 694.454,A -85,B 0,C 180,E1 20850.883,E2 20850.883} C_VEL
LIN {X 0,Y 243.579,Z 689.159,A -85,B 0,C 180,E1 20851.634,E2 20851.634} C_VEL
LIN {X 0,Y 235.048,Z 659.784,A -85,B 0,C 180,E1 20859.259,E2 20859.259} C_VEL
LIN {X 0,Y 224.646,Z 633.028,A -85,B 0,C 180,E1 20867.356,E2 20867.356} C_VEL
LIN {X 0,Y 214.611,Z 611.28,A -85,B 0,C 180,E1 20875.49,E2 20875.49} C_VEL
LIN {X 0,Y 205.049,Z 592.553,A -85,B 0,C 180,E1 20884.508,E2 20884.508} C_VEL
LIN {X 0,Y 199.393,Z 585.258,A -85,B 0,C 180,E1 20890.304,E2 20890.304} C_VEL
LIN {X 0,Y 194.721,Z 578.875,A -85,B 0,C 180,E1 20896.478,E2 20896.478} C_VEL
LIN {X 0,Y 190.364,Z 572.787,A -85,B 0,C 180,E1 20904.575,E2 20904.575} C_VEL
LIN {X 0,Y 186.982,Z 571.056,A -85,B 0,C 180,E1 20915.933,E2 20915.933} C_VEL
LIN {X 0,Y 186.768,Z 571.064,A -85,B 0,C 180,E1 20919.768,E2 20919.768} C_VEL
LIN {X 0,Y 186.507,Z 573.742,A -85,B 0,C 180,E1 20923.715,E2 20923.715} C_VEL
LIN {X 0,Y 186.442,Z 579.608,A -85,B 0,C 180,E1 20929.56,E2 20929.56} C_VEL
LIN {X 0,Y 186.641,Z 579.771,A -85,B 0,C 180,E1 20930.232,E2 20930.232} C_VEL
LIN {X 0,Y 191.628,Z 587.374,A -85,B 0,C 180,E1 20941.704,E2 20941.704} C_VEL
LIN {X 0,Y 199.277,Z 599.479,A -85,B 0,C 180,E1 20952.309,E2 20952.309} C_VEL
LIN {X 0,Y 208.371,Z 616.369,A -85,B 0,C 180,E1 20962.171,E2 20962.171} C_VEL
LIN {X 0,Y 215.165,Z 635.796,A -85,B 0,C 180,E1 20970.002,E2 20970.002} C_VEL
LIN {X 0,Y 220.923,Z 657.246,A -85,B 0,C 180,E1 20977.385,E2 20977.385} C_VEL
LIN {X 0,Y 224.861,Z 680.445,A -85,B 0,C 180,E1 20984.627,E2 20984.627} C_VEL
LIN {X 0,Y 225.304,Z 692.05,A -85,B 0,C 180,E1 20987.99,E2 20987.99} C_VEL
LIN {X 0,Y 208.595,Z 723.899,A -85,B 0,C 180,E1 20994.524,E2 20994.524} C_VEL
LIN {X 0,Y 192.365,Z 751.529,A -85,B 0,C 180,E1 21003.194,E2 21003.194} C_VEL
LIN {X 0,Y 180.614,Z 771.472,A -85,B 0,C 180,E1 21012.785,E2 21012.785} C_VEL
LIN {X 0,Y 172.671,Z 787.014,A -85,B 0,C 180,E1 21024.262,E2 21024.262} C_VEL
LIN {X 0,Y 168.762,Z 797.112,A -85,B 0,C 180,E1 21036.178,E2 21036.178} C_VEL
LIN {X 0,Y 167.964,Z 801.3,A -85,B 0,C 180,E1 21044.299,E2 21044.299} C_VEL
LIN {X 0,Y 169.769,Z 803.821,A -85,B 0,C 180,E1 21054.873,E2 21054.873} C_VEL
LIN {X 0,Y 174.413,Z 803.549,A -85,B 0,C 180,E1 21064.969,E2 21064.969} C_VEL
LIN {X 0,Y 188.119,Z 798.675,A -85,B 0,C 180,E1 21078.769,E2 21078.769} C_VEL
LIN {X 0,Y 216.665,Z 786.415,A -85,B 0,C 180,E1 21092.309,E2 21092.309} C_VEL
LIN {X 0,Y 222.77,Z 783.741,A -85,B 0,C 180,E1 21094.224,E2 21094.224} C_VEL
LIN {X 0,Y 187.077,Z 810.149,A -85,B 0,C 180,E1 21109.647,E2 21109.647} C_VEL
LIN {X 0,Y 172.88,Z 823.857,A -85,B 0,C 180,E1 21124.028,E2 21124.028} C_VEL
LIN {X 0,Y 169.078,Z 829.517,A -85,B 0,C 180,E1 21134.414,E2 21134.414} C_VEL
LIN {X 0,Y 168.6,Z 831.912,A -85,B 0,C 180,E1 21144.846,E2 21144.846} C_VEL
LIN {X 0,Y 169.204,Z 831.767,A -85,B 0,C 180,E1 21149.998,E2 21149.998} C_VEL
LIN {X 0,Y 168.915,Z 828.039,A -85,B 0,C 180,E1 21160.325,E2 21160.325} C_VEL
LIN {X 0,Y 170.789,Z 820,A -85,B 0,C 180,E1 21170.767,E2 21170.767} C_VEL
LIN {X 0,Y 177.327,Z 805.369,A -85,B 0,C 180,E1 21182.249,E2 21182.249} C_VEL
LIN {X 0,Y 189.278,Z 784.157,A -85,B 0,C 180,E1 21192.814,E2 21192.814} C_VEL
LIN {X 0,Y 204.393,Z 757.996,A -85,B 0,C 180,E1 21201.181,E2 21201.181} C_VEL
LIN {X 0,Y 221.499,Z 726.241,A -85,B 0,C 180,E1 21207.765,E2 21207.765} C_VEL
LIN {X 0,Y 237.06,Z 692.381,A -85,B 0,C 180,E1 21212.426,E2 21212.426} C_VEL
LIN {X 0,Y 229.256,Z 663.973,A -85,B 0,C 180,E1 21220.119,E2 21220.119} C_VEL
LIN {X 0,Y 219.886,Z 638.653,A -85,B 0,C 180,E1 21228.087,E2 21228.087} C_VEL
LIN {X 0,Y 210.316,Z 616.908,A -85,B 0,C 180,E1 21236.456,E2 21236.456} C_VEL
LIN {X 0,Y 202.511,Z 601.066,A -85,B 0,C 180,E1 21244.297,E2 21244.297} C_VEL
LIN {X 0,Y 195.755,Z 591.6,A -85,B 0,C 180,E1 21251.759,E2 21251.759} C_VEL
LIN {X 0,Y 192.22,Z 586.279,A -85,B 0,C 180,E1 21256.829,E2 21256.829} C_VEL
LIN {X 0,Y 187.727,Z 579.839,A -85,B 0,C 180,E1 21266.037,E2 21266.037} C_VEL
LIN {X 0,Y 184.615,Z 578.692,A -85,B 0,C 180,E1 21279.781,E2 21279.781} C_VEL
LIN {X 0,Y 186.641,Z 579.771,A -85,B 0,C 180,E1 21290.232,E2 21290.232} C_VEL
LIN {X 0,Y 186.665,Z 583.394,A -85,B 0,C 180,E1 21292.658,E2 21292.658} C_VEL
LIN {X 0,Y 186.013,Z 591.382,A -85,B 0,C 180,E1 21296.049,E2 21296.049} C_VEL
LIN {X 0,Y 186.166,Z 591.753,A -85,B 0,C 180,E1 21296.494,E2 21296.494} C_VEL
LIN {X 0,Y 188.984,Z 595.365,A -85,B 0,C 180,E1 21301.814,E2 21301.814} C_VEL
LIN {X 0,Y 195.244,Z 605.578,A -85,B 0,C 180,E1 21311.139,E2 21311.139} C_VEL
LIN {X 0,Y 202.974,Z 620.422,A -85,B 0,C 180,E1 21320.419,E2 21320.419} C_VEL
LIN {X 0,Y 208.399,Z 635.456,A -85,B 0,C 180,E1 21327.049,E2 21327.049} C_VEL
LIN {X 0,Y 214.172,Z 657.235,A -85,B 0,C 180,E1 21335.071,E2 21335.071} C_VEL
LIN {X 0,Y 218.056,Z 679.935,A -85,B 0,C 180,E1 21342.584,E2 21342.584} C_VEL
LIN {X 0,Y 218.715,Z 693.979,A -85,B 0,C 180,E1 21346.881,E2 21346.881} C_VEL
LIN {X 0,Y 201.672,Z 725.317,A -85,B 0,C 180,E1 21353.475,E2 21353.475} C_VEL
LIN {X 0,Y 185.542,Z 751.798,A -85,B 0,C 180,E1 21361.987,E2 21361.987} C_VEL
LIN {X 0,Y 172.853,Z 772.511,A -85,B 0,C 180,E1 21372.285,E2 21372.285} C_VEL
LIN {X 0,Y 165.089,Z 787.13,A -85,B 0,C 180,E1 21383.394,E2 21383.394} C_VEL
LIN {X 0,Y 161.078,Z 796.986,A -85,B 0,C 180,E1 21395.073,E2 21395.073} C_VEL
LIN {X 0,Y 160.066,Z 801.478,A -85,B 0,C 180,E1 21403.503,E2 21403.503} C_VEL
LIN {X 0,Y 161.792,Z 804.622,A -85,B 0,C 180,E1 21414.619,E2 21414.619} C_VEL
LIN {X 0,Y 167.844,Z 804.592,A -85,B 0,C 180,E1 21427.109,E2 21427.109} C_VEL
LIN {X 0,Y 184.146,Z 799.69,A -85,B 0,C 180,E1 21441.704,E2 21441.704} C_VEL
LIN {X 0,Y 212.244,Z 789.135,A -85,B 0,C 180,E1 21453.922,E2 21453.922} C_VEL
LIN {X 0,Y 208.426,Z 791.795,A -85,B 0,C 180,E1 21455.694,E2 21455.694} C_VEL
LIN {X 0,Y 178.171,Z 812.553,A -85,B 0,C 180,E1 21469.872,E2 21469.872} C_VEL
LIN {X 0,Y 164.14,Z 825.104,A -85,B 0,C 180,E1 21485.472,E2 21485.472} C_VEL
LIN {X 0,Y 160.616,Z 830.377,A -85,B 0,C 180,E1 21499.13,E2 21499.13} C_VEL
LIN {X 0,Y 161.336,Z 830.805,A -85,B 0,C 180,E1 21509.998,E2 21509.998} C_VEL
LIN {X 0,Y 161.103,Z 826.819,A -85,B 0,C 180,E1 21520.831,E2 21520.831} C_VEL
LIN {X 0,Y 163.32,Z 818.268,A -85,B 0,C 180,E1 21532.053,E2 21532.053} C_VEL
LIN {X 0,Y 171.009,Z 802.487,A -85,B 0,C 180,E1 21544.36,E2 21544.36} C_VEL
LIN {X 0,Y 183.924,Z 780.703,A -85,B 0,C 180,E1 21554.981,E2 21554.981} C_VEL
LIN {X 0,Y 200.093,Z 753.676,A -85,B 0,C 180,E1 21563.388,E2 21563.388} C_VEL
LIN {X 0,Y 217.814,Z 721.399,A -85,B 0,C 180,E1 21569.828,E2 21569.828} C_VEL
LIN {X 0,Y 230.231,Z 694.181,A -85,B 0,C 180,E1 21573.612,E2 21573.612} C_VEL
LIN {X 0,Y 222.933,Z 666.658,A -85,B 0,C 180,E1 21581.434,E2 21581.434} C_VEL
LIN {X 0,Y 213.629,Z 640.518,A -85,B 0,C 180,E1 21590.119,E2 21590.119} C_VEL
LIN {X 0,Y 204.58,Z 619.382,A -85,B 0,C 180,E1 21598.949,E2 21598.949} C_VEL
LIN {X 0,Y 197.988,Z 605.806,A -85,B 0,C 180,E1 21606.223,E2 21606.223} C_VEL
LIN {X 0,Y 190.9,Z 595.537,A -85,B 0,C 180,E1 21615.194,E2 21615.194} C_VEL
LIN {X 0,Y 185.5,Z 587.412,A -85,B 0,C 180,E1 21626.131,E2 21626.131} C_VEL
LIN {X 0,Y 182.763,Z 586.293,A -85,B 0,C 180,E1 21635.455,E2 21635.455} C_VEL
LIN {X 0,Y 183.837,Z 587.162,A -85,B 0,C 180,E1 21648.789,E2 21648.789} C_VEL
LIN {X 0,Y 184.67,Z 587.785,A -85,B 0,C 180,E1 21651.491,E2 21651.491} C_VEL
LIN {X 0,Y 186.166,Z 591.753,A -85,B 0,C 180,E1 21656.494,E2 21656.494} C_VEL
LIN {X 0,Y 187.12,Z 596.79,A -85,B 0,C 180,E1 21660.203,E2 21660.203} C_VEL
LIN {X 0,Y 188.294,Z 606.487,A -85,B 0,C 180,E1 21665.526,E2 21665.526} C_VEL
LIN {X 0,Y 188.713,Z 607.109,A -85,B 0,C 180,E1 21666.159,E2 21666.159} C_VEL
LIN {X 0,Y 195.284,Z 619.466,A -85,B 0,C 180,E1 21675.552,E2 21675.552} C_VEL
LIN {X 0,Y 201.096,Z 632.909,A -85,B 0,C 180,E1 21682.889,E2 21682.889} C_VEL
LIN {X 0,Y 206.863,Z 654.643,A -85,B 0,C 180,E1 21691.673,E2 21691.673} C_VEL
LIN {X 0,Y 210.859,Z 676.592,A -85,B 0,C 180,E1 21699.43,E2 21699.43} C_VEL
LIN {X 0,Y 212.528,Z 694.746,A -85,B 0,C 180,E1 21705.47,E2 21705.47} C_VEL
LIN {X 0,Y 195.091,Z 726.179,A -85,B 0,C 180,E1 21712.23,E2 21712.23} C_VEL
LIN {X 0,Y 178.357,Z 752.701,A -85,B 0,C 180,E1 21720.975,E2 21720.975} C_VEL
LIN {X 0,Y 165.152,Z 773.466,A -85,B 0,C 180,E1 21731.687,E2 21731.687} C_VEL
LIN {X 0,Y 157.145,Z 788.006,A -85,B 0,C 180,E1 21743.281,E2 21743.281} C_VEL
LIN {X 0,Y 153.281,Z 797.177,A -85,B 0,C 180,E1 21754.505,E2 21754.505} C_VEL
LIN {X 0,Y 152.529,Z 803.816,A -85,B 0,C 180,E1 21768.537,E2 21768.537} C_VEL
LIN {X 0,Y 155.86,Z 805.961,A -85,B 0,C 180,E1 21779.988,E2 21779.988} C_VEL
LIN {X 0,Y 167.641,Z 804.447,A -85,B 0,C 180,E1 21795.709,E2 21795.709} C_VEL
LIN {X 0,Y 193.767,Z 796.613,A -85,B 0,C 180,E1 21810.733,E2 21810.733} C_VEL
LIN {X 0,Y 202.035,Z 794.169,A -85,B 0,C 180,E1 21814.474,E2 21814.474} C_VEL
LIN {X 0,Y 170.043,Z 814.024,A -85,B 0,C 180,E1 21829.51,E2 21829.51} C_VEL
LIN {X 0,Y 156.719,Z 824.583,A -85,B 0,C 180,E1 21844.228,E2 21844.228} C_VEL
LIN {X 0,Y 152.76,Z 829.601,A -85,B 0,C 180,E1 21858.564,E2 21858.564} C_VEL
LIN {X 0,Y 153.485,Z 829.76,A -85,B 0,C 180,E1 21869.998,E2 21869.998} C_VEL
LIN {X 0,Y 153.277,Z 825.565,A -85,B 0,C 180,E1 21881.392,E2 21881.392} C_VEL
LIN {X 0,Y 155.714,Z 816.98,A -85,B 0,C 180,E1 21892.886,E2 21892.886} C_VEL
LIN {X 0,Y 163.635,Z 801.57,A -85,B 0,C 180,E1 21905.328,E2 21905.328} C_VEL
LIN {X 0,Y 177.007,Z 779.992,A -85,B 0,C 180,E1 21916.19,E2 21916.19} C_VEL
LIN {X 0,Y 193.769,Z 753.01,A -85,B 0,C 180,E1 21924.765,E2 21924.765} C_VEL
LIN {X 0,Y 212.367,Z 720.122,A -85,B 0,C 180,E1 21931.376,E2 21931.376} C_VEL
LIN {X 0,Y 223.488,Z 696.363,A -85,B 0,C 180,E1 21934.761,E2 21934.761} C_VEL
LIN {X 0,Y 216.725,Z 669.633,A -85,B 0,C 180,E1 21942.737,E2 21942.737} C_VEL
LIN {X 0,Y 208.544,Z 645.473,A -85,B 0,C 180,E1 21951.134,E2 21951.134} C_VEL
LIN {X 0,Y 200.182,Z 624.91,A -85,B 0,C 180,E1 21960.009,E2 21960.009} C_VEL
LIN {X 0,Y 194.95,Z 613.331,A -85,B 0,C 180,E1 21966.32,E2 21966.32} C_VEL
LIN {X 0,Y 187.637,Z 602.08,A -85,B 0,C 180,E1 21976.273,E2 21976.273} C_VEL
LIN {X 0,Y 183.377,Z 596.137,A -85,B 0,C 180,E1 21984.744,E2 21984.744} C_VEL
LIN {X 0,Y 180.769,Z 593.913,A -85,B 0,C 180,E1 21993.12,E2 21993.12} C_VEL
LIN {X 0,Y 181.145,Z 594.554,A -85,B 0,C 180,E1 22008.039,E2 22008.039} C_VEL
LIN {X 0,Y 182.347,Z 596.959,A -85,B 0,C 180,E1 22013.037,E2 22013.037} C_VEL
LIN {X 0,Y 186.116,Z 602.981,A -85,B 0,C 180,E1 22021.768,E2 22021.768} C_VEL
LIN {X 0,Y 188.713,Z 607.109,A -85,B 0,C 180,E1 22026.159,E2 22026.159} C_VEL
LIN {X 0,Y 190.122,Z 613.172,A -85,B 0,C 180,E1 22029.626,E2 22029.626} C_VEL
LIN {X 0,Y 191.348,Z 626.15,A -85,B 0,C 180,E1 22035.073,E2 22035.073} C_VEL
LIN {X 0,Y 196.745,Z 639.911,A -85,B 0,C 180,E1 22042.731,E2 22042.731} C_VEL
LIN {X 0,Y 201.775,Z 661.41,A -85,B 0,C 180,E1 22051.614,E2 22051.614} C_VEL
LIN {X 0,Y 204.948,Z 683.261,A -85,B 0,C 180,E1 22059.57,E2 22059.57} C_VEL
LIN {X 0,Y 205.945,Z 697.133,A -85,B 0,C 180,E1 22064.36,E2 22064.36} C_VEL
LIN {X 0,Y 187.468,Z 728.766,A -85,B 0,C 180,E1 22071.387,E2 22071.387} C_VEL
LIN {X 0,Y 170.335,Z 754.832,A -85,B 0,C 180,E1 22080.448,E2 22080.448} C_VEL
LIN {X 0,Y 156.968,Z 775.113,A -85,B 0,C 180,E1 22091.565,E2 22091.565} C_VEL
LIN {X 0,Y 148.535,Z 790.198,A -85,B 0,C 180,E1 22104.638,E2 22104.638} C_VEL
LIN {X 0,Y 145.162,Z 798.254,A -85,B 0,C 180,E1 22115.329,E2 22115.329} C_VEL
LIN {X 0,Y 144.531,Z 804.157,A -85,B 0,C 180,E1 22127.894,E2 22127.894} C_VEL
LIN {X 0,Y 147.881,Z 806.778,A -85,B 0,C 180,E1 22139.988,E2 22139.988} C_VEL
LIN {X 0,Y 160.171,Z 806.053,A -85,B 0,C 180,E1 22156.462,E2 22156.462} C_VEL
LIN {X 0,Y 187.376,Z 799.445,A -85,B 0,C 180,E1 22171.902,E2 22171.902} C_VEL
LIN {X 0,Y 192.494,Z 797.996,A -85,B 0,C 180,E1 22173.86,E2 22173.86} C_VEL
LIN {X 0,Y 158.752,Z 817.405,A -85,B 0,C 180,E1 22191.686,E2 22191.686} C_VEL
LIN {X 0,Y 147.073,Z 826.147,A -85,B 0,C 180,E1 22207.862,E2 22207.862} C_VEL
LIN {X 0,Y 144.927,Z 828.723,A -85,B 0,C 180,E1 22217.937,E2 22217.937} C_VEL
LIN {X 0,Y 145.64,Z 828.695,A -85,B 0,C 180,E1 22229.997,E2 22229.997} C_VEL
LIN {X 0,Y 145.483,Z 824.298,A -85,B 0,C 180,E1 22242.011,E2 22242.011} C_VEL
LIN {X 0,Y 148.248,Z 815.32,A -85,B 0,C 180,E1 22254.109,E2 22254.109} C_VEL
LIN {X 0,Y 156.975,Z 799.498,A -85,B 0,C 180,E1 22267.07,E2 22267.07} C_VEL
LIN {X 0,Y 170.462,Z 778.772,A -85,B 0,C 180,E1 22277.667,E2 22277.667} C_VEL
LIN {X 0,Y 187.107,Z 753.014,A -85,B 0,C 180,E1 22286.036,E2 22286.036} C_VEL
LIN {X 0,Y 206.099,Z 720.612,A -85,B 0,C 180,E1 22292.689,E2 22292.689} C_VEL
LIN {X 0,Y 216.801,Z 698.632,A -85,B 0,C 180,E1 22295.922,E2 22295.922} C_VEL
LIN {X 0,Y 210.757,Z 673.257,A -85,B 0,C 180,E1 22303.846,E2 22303.846} C_VEL
LIN {X 0,Y 202.929,Z 648.974,A -85,B 0,C 180,E1 22312.735,E2 22312.735} C_VEL
LIN {X 0,Y 195.207,Z 628.796,A -85,B 0,C 180,E1 22321.903,E2 22321.903} C_VEL
LIN {X 0,Y 189.663,Z 617.256,A -85,B 0,C 180,E1 22329.197,E2 22329.197} C_VEL
LIN {X 0,Y 184.26,Z 608.593,A -85,B 0,C 180,E1 22337.364,E2 22337.364} C_VEL
LIN {X 0,Y 179.53,Z 602.439,A -85,B 0,C 180,E1 22348.196,E2 22348.196} C_VEL
LIN {X 0,Y 177.469,Z 601.29,A -85,B 0,C 180,E1 22359.844,E2 22359.844} C_VEL
LIN {X 0,Y 179.326,Z 603.214,A -85,B 0,C 180,E1 22371.497,E2 22371.497} C_VEL
LIN {X 0,Y 182.956,Z 610.142,A -85,B 0,C 180,E1 22381.379,E2 22381.379} C_VEL
LIN {X 0,Y 188.364,Z 619.989,A -85,B 0,C 180,E1 22390.752,E2 22390.752} C_VEL
LIN {X 0,Y 191.348,Z 626.15,A -85,B 0,C 180,E1 22395.073,E2 22395.073} C_VEL
LIN {X 0,Y 192.495,Z 633.631,A -85,B 0,C 180,E1 22398.277,E2 22398.277} C_VEL
LIN {X 0,Y 192.574,Z 648.444,A -85,B 0,C 180,E1 22403.269,E2 22403.269} C_VEL
LIN {X 0,Y 196.78,Z 669.792,A -85,B 0,C 180,E1 22412.209,E2 22412.209} C_VEL
LIN {X 0,Y 199.062,Z 691.679,A -85,B 0,C 180,E1 22420.409,E2 22420.409} C_VEL
LIN {X 0,Y 198.772,Z 700.228,A -85,B 0,C 180,E1 22423.305,E2 22423.305} C_VEL
LIN {X 0,Y 179.461,Z 731.751,A -85,B 0,C 180,E1 22430.631,E2 22430.631} C_VEL
LIN {X 0,Y 163.04,Z 755.893,A -85,B 0,C 180,E1 22439.408,E2 22439.408} C_VEL
LIN {X 0,Y 149.052,Z 776.36,A -85,B 0,C 180,E1 22451.155,E2 22451.155} C_VEL
LIN {X 0,Y 140.463,Z 791.244,A -85,B 0,C 180,E1 22464.859,E2 22464.859} C_VEL
LIN {X 0,Y 136.884,Z 799.894,A -85,B 0,C 180,E1 22477.21,E2 22477.21} C_VEL
LIN {X 0,Y 137.728,Z 806.344,A -85,B 0,C 180,E1 22493.676,E2 22493.676} C_VEL
LIN {X 0,Y 143.067,Z 808.146,A -85,B 0,C 180,E1 22506.062,E2 22506.062} C_VEL
LIN {X 0,Y 159.343,Z 806.637,A -85,B 0,C 180,E1 22522.325,E2 22522.325} C_VEL
LIN {X 0,Y 182.673,Z 801.824,A -85,B 0,C 180,E1 22534.017,E2 22534.017} C_VEL
LIN {X 0,Y 152.401,Z 817.324,A -85,B 0,C 180,E1 22549.774,E2 22549.774} C_VEL
LIN {X 0,Y 140.505,Z 824.785,A -85,B 0,C 180,E1 22564.464,E2 22564.464} C_VEL
LIN {X 0,Y 137.102,Z 827.843,A -85,B 0,C 180,E1 22577.237,E2 22577.237} C_VEL
LIN {X 0,Y 137.781,Z 827.619,A -85,B 0,C 180,E1 22589.997,E2 22589.997} C_VEL
LIN {X 0,Y 137.705,Z 822.975,A -85,B 0,C 180,E1 22602.7,E2 22602.7} C_VEL
LIN {X 0,Y 141.6,Z 812.219,A -85,B 0,C 180,E1 22617.025,E2 22617.025} C_VEL
LIN {X 0,Y 151.916,Z 795.229,A -85,B 0,C 180,E1 22630.374,E2 22630.374} C_VEL
LIN {X 0,Y 167.874,Z 771.83,A -85,B 0,C 180,E1 22641.488,E2 22641.488} C_VEL
LIN {X 0,Y 186.357,Z 743.687,A -85,B 0,C 180,E1 22649.678,E2 22649.678} C_VEL
LIN {X 0,Y 205.409,Z 710.862,A -85,B 0,C 180,E1 22655.628,E2 22655.628} C_VEL
LIN {X 0,Y 210.103,Z 700.732,A -85,B 0,C 180,E1 22657.132,E2 22657.132} C_VEL
LIN {X 0,Y 204.729,Z 676.782,A -85,B 0,C 180,E1 22665.008,E2 22665.008} C_VEL
LIN {X 0,Y 197.826,Z 654.038,A -85,B 0,C 180,E1 22673.697,E2 22673.697} C_VEL
LIN {X 0,Y 190.982,Z 634.693,A -85,B 0,C 180,E1 22682.85,E2 22682.85} C_VEL
LIN {X 0,Y 185.674,Z 623.336,A -85,B 0,C 180,E1 22690.303,E2 22690.303} C_VEL
LIN {X 0,Y 180.115,Z 614.778,A -85,B 0,C 180,E1 22699.658,E2 22699.658} C_VEL
LIN {X 0,Y 177.862,Z 611.031,A -85,B 0,C 180,E1 22705.201,E2 22705.201} C_VEL
LIN {X 0,Y 176.05,Z 609.064,A -85,B 0,C 180,E1 22711.076,E2 22711.076} C_VEL
LIN {X 0,Y 175.365,Z 609.195,A -85,B 0,C 180,E1 22726.317,E2 22726.317} C_VEL
LIN {X 0,Y 176.32,Z 610.27,A -85,B 0,C 180,E1 22730.623,E2 22730.623} C_VEL
LIN {X 0,Y 179.804,Z 617.573,A -85,B 0,C 180,E1 22741.321,E2 22741.321} C_VEL
LIN {X 0,Y 184.004,Z 625.715,A -85,B 0,C 180,E1 22749.387,E2 22749.387} C_VEL
LIN {X 0,Y 190.029,Z 639.429,A -85,B 0,C 180,E1 22758.757,E2 22758.757} C_VEL
LIN {X 0,Y 192.574,Z 648.444,A -85,B 0,C 180,E1 22763.269,E2 22763.269} C_VEL
LIN {X 0,Y 192.539,Z 657.242,A -85,B 0,C 180,E1 22766.165,E2 22766.165} C_VEL
LIN {X 0,Y 190.774,Z 672.952,A -85,B 0,C 180,E1 22770.824,E2 22770.824} C_VEL
LIN {X 0,Y 192.681,Z 695.301,A -85,B 0,C 180,E1 22779.575,E2 22779.575} C_VEL
LIN {X 0,Y 192.205,Z 702.277,A -85,B 0,C 180,E1 22781.993,E2 22781.993} C_VEL
LIN {X 0,Y 172.764,Z 732.918,A -85,B 0,C 180,E1 22789.277,E2 22789.277} C_VEL
LIN {X 0,Y 155.251,Z 757.62,A -85,B 0,C 180,E1 22798.611,E2 22798.611} C_VEL
LIN {X 0,Y 140.738,Z 778.092,A -85,B 0,C 180,E1 22811.126,E2 22811.126} C_VEL
LIN {X 0,Y 132.343,Z 792.258,A -85,B 0,C 180,E1 22825.093,E2 22825.093} C_VEL
LIN {X 0,Y 128.735,Z 801.38,A -85,B 0,C 180,E1 22839.325,E2 22839.325} C_VEL
LIN {X 0,Y 130.284,Z 807.219,A -85,B 0,C 180,E1 22855.784,E2 22855.784} C_VEL
LIN {X 0,Y 139.589,Z 809.347,A -85,B 0,C 180,E1 22872.515,E2 22872.515} C_VEL
LIN {X 0,Y 160.219,Z 807.259,A -85,B 0,C 180,E1 22888.183,E2 22888.183} C_VEL
LIN {X 0,Y 171.7,Z 805.282,A -85,B 0,C 180,E1 22893.35,E2 22893.35} C_VEL
LIN {X 0,Y 165.186,Z 808.377,A -85,B 0,C 180,E1 22896.827,E2 22896.827} C_VEL
LIN {X 0,Y 139.194,Z 820.72,A -85,B 0,C 180,E1 22914.187,E2 22914.187} C_VEL
LIN {X 0,Y 130.569,Z 825.938,A -85,B 0,C 180,E1 22929.639,E2 22929.639} C_VEL
LIN {X 0,Y 129.154,Z 827.182,A -85,B 0,C 180,E1 22943.265,E2 22943.265} C_VEL
LIN {X 0,Y 129.937,Z 826.526,A -85,B 0,C 180,E1 22949.997,E2 22949.997} C_VEL
LIN {X 0,Y 129.943,Z 821.53,A -85,B 0,C 180,E1 22963.473,E2 22963.473} C_VEL
LIN {X 0,Y 134.392,Z 810.383,A -85,B 0,C 180,E1 22978.604,E2 22978.604} C_VEL
LIN {X 0,Y 145.043,Z 793.867,A -85,B 0,C 180,E1 22991.895,E2 22991.895} C_VEL
LIN {X 0,Y 161.733,Z 770.486,A -85,B 0,C 180,E1 23003.229,E2 23003.229} C_VEL
LIN {X 0,Y 180.921,Z 742.274,A -85,B 0,C 180,E1 23011.483,E2 23011.483} C_VEL
LIN {X 0,Y 200.708,Z 709.026,A -85,B 0,C 180,E1 23017.452,E2 23017.452} C_VEL
LIN {X 0,Y 203.328,Z 703.974,A -85,B 0,C 180,E1 23018.151,E2 23018.151} C_VEL
LIN {X 0,Y 199.169,Z 682.107,A -85,B 0,C 180,E1 23025.566,E2 23025.566} C_VEL
LIN {X 0,Y 193.016,Z 660.03,A -85,B 0,C 180,E1 23034.283,E2 23034.283} C_VEL
LIN {X 0,Y 186.755,Z 640.941,A -85,B 0,C 180,E1 23043.556,E2 23043.556} C_VEL
LIN {X 0,Y 182.308,Z 630.557,A -85,B 0,C 180,E1 23050.495,E2 23050.495} C_VEL
LIN {X 0,Y 176.896,Z 621.887,A -85,B 0,C 180,E1 23060.031,E2 23060.031} C_VEL
LIN {X 0,Y 173.582,Z 616.967,A -85,B 0,C 180,E1 23069.284,E2 23069.284} C_VEL
LIN {X 0,Y 171.975,Z 616.086,A -85,B 0,C 180,E1 23078.057,E2 23078.057} C_VEL
LIN {X 0,Y 172.699,Z 616.977,A -85,B 0,C 180,E1 23088.134,E2 23088.134} C_VEL
LIN {X 0,Y 176.196,Z 624.299,A -85,B 0,C 180,E1 23100.677,E2 23100.677} C_VEL
LIN {X 0,Y 180.139,Z 632.464,A -85,B 0,C 180,E1 23108.924,E2 23108.924} C_VEL
LIN {X 0,Y 185.16,Z 644.84,A -85,B 0,C 180,E1 23117.751,E2 23117.751} C_VEL
LIN {X 0,Y 188.384,Z 658.473,A -85,B 0,C 180,E1 23124.565,E2 23124.565} C_VEL
LIN {X 0,Y 190.774,Z 672.952,A -85,B 0,C 180,E1 23130.824,E2 23130.824} C_VEL
LIN {X 0,Y 189.769,Z 682.145,A -85,B 0,C 180,E1 23133.66,E2 23133.66} C_VEL
LIN {X 0,Y 186.272,Z 697.853,A -85,B 0,C 180,E1 23138.288,E2 23138.288} C_VEL
LIN {X 0,Y 186.172,Z 703.449,A -85,B 0,C 180,E1 23140.456,E2 23140.456} C_VEL
LIN {X 0,Y 165.843,Z 734.358,A -85,B 0,C 180,E1 23147.937,E2 23147.937} C_VEL
LIN {X 0,Y 146.61,Z 760.544,A -85,B 0,C 180,E1 23158.37,E2 23158.37} C_VEL
LIN {X 0,Y 132.208,Z 780.159,A -85,B 0,C 180,E1 23171.384,E2 23171.384} C_VEL
LIN {X 0,Y 123.845,Z 794.032,A -85,B 0,C 180,E1 23186.432,E2 23186.432} C_VEL
LIN {X 0,Y 120.604,Z 803.154,A -85,B 0,C 180,E1 23202.445,E2 23202.445} C_VEL
LIN {X 0,Y 123.887,Z 808.709,A -85,B 0,C 180,E1 23219.985,E2 23219.985} C_VEL
LIN {X 0,Y 137.859,Z 810.47,A -85,B 0,C 180,E1 23239.223,E2 23239.223} C_VEL
LIN {X 0,Y 161.771,Z 808.147,A -85,B 0,C 180,E1 23253.343,E2 23253.343} C_VEL
LIN {X 0,Y 160.845,Z 808.732,A -85,B 0,C 180,E1 23254.373,E2 23254.373} C_VEL
LIN {X 0,Y 130.5,Z 821.368,A -85,B 0,C 180,E1 23274.539,E2 23274.539} C_VEL
LIN {X 0,Y 121.497,Z 826.075,A -85,B 0,C 180,E1 23295.565,E2 23295.565} C_VEL
LIN {X 0,Y 122.078,Z 825.388,A -85,B 0,C 180,E1 23309.997,E2 23309.997} C_VEL
LIN {X 0,Y 122.197,Z 820.036,A -85,B 0,C 180,E1 23324.345,E2 23324.345} C_VEL
LIN {X 0,Y 126.36,Z 810.134,A -85,B 0,C 180,E1 23338.635,E2 23338.635} C_VEL
LIN {X 0,Y 137.535,Z 793.506,A -85,B 0,C 180,E1 23352.897,E2 23352.897} C_VEL
LIN {X 0,Y 154.464,Z 770.824,A -85,B 0,C 180,E1 23364.421,E2 23364.421} C_VEL
LIN {X 0,Y 174.127,Z 743.038,A -85,B 0,C 180,E1 23372.839,E2 23372.839} C_VEL
LIN {X 0,Y 194.684,Z 709.721,A -85,B 0,C 180,E1 23378.941,E2 23378.941} C_VEL
LIN {X 0,Y 196.694,Z 704.6,A -85,B 0,C 180,E1 23379.899,E2 23379.899} C_VEL
LIN {X 0,Y 192.32,Z 682.238,A -85,B 0,C 180,E1 23388.084,E2 23388.084} C_VEL
LIN {X 0,Y 186.327,Z 659.773,A -85,B 0,C 180,E1 23397.708,E2 23397.708} C_VEL
LIN {X 0,Y 180.972,Z 642.65,A -85,B 0,C 180,E1 23407,E2 23407} C_VEL
LIN {X 0,Y 176.15,Z 633.448,A -85,B 0,C 180,E1 23414.953,E2 23414.953} C_VEL
LIN {X 0,Y 172.152,Z 626.772,A -85,B 0,C 180,E1 23424,E2 23424} C_VEL
LIN {X 0,Y 169.852,Z 623.683,A -85,B 0,C 180,E1 23432.345,E2 23432.345} C_VEL
LIN {X 0,Y 169.253,Z 623.768,A -85,B 0,C 180,E1 23445.71,E2 23445.71} C_VEL
LIN {X 0,Y 171.015,Z 627.966,A -85,B 0,C 180,E1 23455.4,E2 23455.4} C_VEL
LIN {X 0,Y 174.268,Z 634.576,A -85,B 0,C 180,E1 23464.255,E2 23464.255} C_VEL
LIN {X 0,Y 179.151,Z 646.878,A -85,B 0,C 180,E1 23474.436,E2 23474.436} C_VEL
LIN {X 0,Y 182.291,Z 658.271,A -85,B 0,C 180,E1 23481.125,E2 23481.125} C_VEL
LIN {X 0,Y 185.14,Z 679.028,A -85,B 0,C 180,E1 23490.588,E2 23490.588} C_VEL
LIN {X 0,Y 186.272,Z 697.853,A -85,B 0,C 180,E1 23498.288,E2 23498.288} C_VEL
LIN {X 0,Y 183.92,Z 703.129,A -85,B 0,C 180,E1 23499.527,E2 23499.527} C_VEL
LIN {X 0,Y 173.227,Z 715.55,A -85,B 0,C 180,E1 23501.11,E2 23501.11} C_VEL
LIN {X 0,Y 153.709,Z 742.938,A -85,B 0,C 180,E1 23508.913,E2 23508.913} C_VEL
LIN {X 0,Y 135.288,Z 766.667,A -85,B 0,C 180,E1 23520.092,E2 23520.092} C_VEL
LIN {X 0,Y 121.714,Z 784.743,A -85,B 0,C 180,E1 23534.317,E2 23534.317} C_VEL
LIN {X 0,Y 114.601,Z 797.166,A -85,B 0,C 180,E1 23550.284,E2 23550.284} C_VEL
LIN {X 0,Y 112.678,Z 804.242,A -85,B 0,C 180,E1 23564.394,E2 23564.394} C_VEL
LIN {X 0,Y 115.876,Z 809.153,A -85,B 0,C 180,E1 23579.984,E2 23579.984} C_VEL
LIN {X 0,Y 130.485,Z 811.761,A -85,B 0,C 180,E1 23600.356,E2 23600.356} C_VEL
LIN {X 0,Y 151.319,Z 810.641,A -85,B 0,C 180,E1 23613.169,E2 23613.169} C_VEL
LIN {X 0,Y 148.34,Z 811.951,A -85,B 0,C 180,E1 23615.256,E2 23615.256} C_VEL
LIN {X 0,Y 121.198,Z 821.951,A -85,B 0,C 180,E1 23635.791,E2 23635.791} C_VEL
LIN {X 0,Y 113.757,Z 825.067,A -85,B 0,C 180,E1 23654.559,E2 23654.559} C_VEL
LIN {X 0,Y 114.257,Z 824.129,A -85,B 0,C 180,E1 23669.997,E2 23669.997} C_VEL
LIN {X 0,Y 114.486,Z 818.527,A -85,B 0,C 180,E1 23685.334,E2 23685.334} C_VEL
LIN {X 0,Y 119.287,Z 808.149,A -85,B 0,C 180,E1 23700.508,E2 23700.508} C_VEL
LIN {X 0,Y 131.217,Z 791.545,A -85,B 0,C 180,E1 23715.014,E2 23715.014} C_VEL
LIN {X 0,Y 149.29,Z 768.415,A -85,B 0,C 180,E1 23726.788,E2 23726.788} C_VEL
LIN {X 0,Y 169.072,Z 741.413,A -85,B 0,C 180,E1 23734.864,E2 23734.864} C_VEL
LIN {X 0,Y 189.473,Z 709.172,A -85,B 0,C 180,E1 23740.711,E2 23740.711} C_VEL
LIN {X 0,Y 189.795,Z 704.634,A -85,B 0,C 180,E1 23742.094,E2 23742.094} C_VEL
LIN {X 0,Y 185.952,Z 684.173,A -85,B 0,C 180,E1 23750.047,E2 23750.047} C_VEL
LIN {X 0,Y 181.009,Z 663.897,A -85,B 0,C 180,E1 23759.23,E2 23759.23} C_VEL
LIN {X 0,Y 176.209,Z 647.499,A -85,B 0,C 180,E1 23768.658,E2 23768.658} C_VEL
LIN {X 0,Y 171.309,Z 637.72,A -85,B 0,C 180,E1 23778.127,E2 23778.127} C_VEL
LIN {X 0,Y 168.109,Z 632.354,A -85,B 0,C 180,E1 23786.776,E2 23786.776} C_VEL
LIN {X 0,Y 166.08,Z 630.748,A -85,B 0,C 180,E1 23794.871,E2 23794.871} C_VEL
LIN {X 0,Y 166.067,Z 631.368,A -85,B 0,C 180,E1 23806.848,E2 23806.848} C_VEL
LIN {X 0,Y 168.223,Z 636.17,A -85,B 0,C 180,E1 23817.318,E2 23817.318} C_VEL
LIN {X 0,Y 171.217,Z 643.819,A -85,B 0,C 180,E1 23826.165,E2 23826.165} C_VEL
LIN {X 0,Y 175.128,Z 654.711,A -85,B 0,C 180,E1 23834.97,E2 23834.97} C_VEL
LIN {X 0,Y 177.5,Z 666.351,A -85,B 0,C 180,E1 23841.631,E2 23841.631} C_VEL
LIN {X 0,Y 179.435,Z 685.589,A -85,B 0,C 180,E1 23850.606,E2 23850.606} C_VEL
LIN {X 0,Y 179.851,Z 704.151,A -85,B 0,C 180,E1 23858.474,E2 23858.474} C_VEL
LIN {X 0,Y 176.144,Z 711.144,A -85,B 0,C 180,E1 23860.122,E2 23860.122} C_VEL
LIN {X 0,Y 173.227,Z 715.55,A -85,B 0,C 180,E1 23861.11,E2 23861.11} C_VEL
LIN {X 0,Y 168.151,Z 721.872,A -85,B 0,C 180,E1 23862.283,E2 23862.283} C_VEL
LIN {X 0,Y 151.825,Z 737.808,A -85,B 0,C 180,E1 23865.172,E2 23865.172} C_VEL
LIN {X 0,Y 150.672,Z 739.244,A -85,B 0,C 180,E1 23865.624,E2 23865.624} C_VEL
LIN {X 0,Y 129.77,Z 765.249,A -85,B 0,C 180,E1 23877.365,E2 23877.365} C_VEL
LIN {X 0,Y 114.729,Z 784.234,A -85,B 0,C 180,E1 23892.372,E2 23892.372} C_VEL
LIN {X 0,Y 107.387,Z 796.204,A -85,B 0,C 180,E1 23907.78,E2 23907.78} C_VEL
LIN {X 0,Y 104.939,Z 805.633,A -85,B 0,C 180,E1 23927.484,E2 23927.484} C_VEL
LIN {X 0,Y 111.495,Z 811.099,A -85,B 0,C 180,E1 23947.788,E2 23947.788} C_VEL
LIN {X 0,Y 131.103,Z 812.976,A -85,B 0,C 180,E1 23967.496,E2 23967.496} C_VEL
LIN {X 0,Y 141.338,Z 812.663,A -85,B 0,C 180,E1 23973.196,E2 23973.196} C_VEL
LIN {X 0,Y 116.281,Z 820.764,A -85,B 0,C 180,E1 23991.348,E2 23991.348} C_VEL
LIN {X 0,Y 106.025,Z 824.021,A -85,B 0,C 180,E1 24013.401,E2 24013.401} C_VEL
LIN {X 0,Y 106.442,Z 822.862,A -85,B 0,C 180,E1 24029.996,E2 24029.996} C_VEL
LIN {X 0,Y 106.822,Z 816.97,A -85,B 0,C 180,E1 24046.464,E2 24046.464} C_VEL
LIN {X 0,Y 113.29,Z 804.77,A -85,B 0,C 180,E1 24064.23,E2 24064.23} C_VEL
LIN {X 0,Y 128.696,Z 785.249,A -85,B 0,C 180,E1 24080.092,E2 24080.092} C_VEL
LIN {X 0,Y 148.863,Z 760.243,A -85,B 0,C 180,E1 24091.306,E2 24091.306} C_VEL
LIN {X 0,Y 170.184,Z 730.912,A -85,B 0,C 180,E1 24098.86,E2 24098.86} C_VEL
LIN {X 0,Y 183.545,Z 709.468,A -85,B 0,C 180,E1 24102.532,E2 24102.532} C_VEL
LIN {X 0,Y 180.205,Z 688.75,A -85,B 0,C 180,E1 24110.947,E2 24110.947} C_VEL
LIN {X 0,Y 175.843,Z 668.461,A -85,B 0,C 180,E1 24120.627,E2 24120.627} C_VEL
LIN {X 0,Y 172.123,Z 654.282,A -85,B 0,C 180,E1 24129.031,E2 24129.031} C_VEL
LIN {X 0,Y 167.628,Z 644.691,A -85,B 0,C 180,E1 24138.44,E2 24138.44} C_VEL
LIN {X 0,Y 164.565,Z 639.354,A -85,B 0,C 180,E1 24147.4,E2 24147.4} C_VEL
LIN {X 0,Y 162.976,Z 637.988,A -85,B 0,C 180,E1 24153.889,E2 24153.889} C_VEL
LIN {X 0,Y 162.295,Z 637.866,A -85,B 0,C 180,E1 24161.73,E2 24161.73} C_VEL
LIN {X 0,Y 162.973,Z 639.332,A -85,B 0,C 180,E1 24169.437,E2 24169.437} C_VEL
LIN {X 0,Y 165.062,Z 644.77,A -85,B 0,C 180,E1 24179.277,E2 24179.277} C_VEL
LIN {X 0,Y 168.321,Z 653.866,A -85,B 0,C 180,E1 24188.914,E2 24188.914} C_VEL
LIN {X 0,Y 171.647,Z 666.248,A -85,B 0,C 180,E1 24197.908,E2 24197.908} C_VEL
LIN {X 0,Y 173.317,Z 685.189,A -85,B 0,C 180,E1 24207.499,E2 24207.499} C_VEL
LIN {X 0,Y 173.516,Z 704.931,A -85,B 0,C 180,E1 24216.376,E2 24216.376} C_VEL
LIN {X 0,Y 172.864,Z 708.132,A -85,B 0,C 180,E1 24217.57,E2 24217.57} C_VEL
LIN {X 0,Y 151.477,Z 738.182,A -85,B 0,C 180,E1 24225.27,E2 24225.27} C_VEL
LIN {X 0,Y 150.672,Z 739.244,A -85,B 0,C 180,E1 24225.624,E2 24225.624} C_VEL
LIN {X 0,Y 139.167,Z 750.063,A -85,B 0,C 180,E1 24228.644,E2 24228.644} C_VEL
LIN {X 0,Y 127.665,Z 760.086,A -85,B 0,C 180,E1 24232.388,E2 24232.388} C_VEL
LIN {X 0,Y 109.973,Z 781.019,A -85,B 0,C 180,E1 24247.519,E2 24247.519} C_VEL
LIN {X 0,Y 100.064,Z 795.356,A -85,B 0,C 180,E1 24265.587,E2 24265.587} C_VEL
LIN {X 0,Y 96.94,Z 803.545,A -85,B 0,C 180,E1 24281.778,E2 24281.778} C_VEL
LIN {X 0,Y 99.744,Z 809.63,A -85,B 0,C 180,E1 24299.982,E2 24299.982} C_VEL
LIN {X 0,Y 115.857,Z 813.882,A -85,B 0,C 180,E1 24323.065,E2 24323.065} C_VEL
LIN {X 0,Y 130.988,Z 814.307,A -85,B 0,C 180,E1 24333.079,E2 24333.079} C_VEL
LIN {X 0,Y 105.156,Z 821.43,A -85,B 0,C 180,E1 24354.831,E2 24354.831} C_VEL
LIN {X 0,Y 98.357,Z 822.971,A -85,B 0,C 180,E1 24372.065,E2 24372.065} C_VEL
LIN {X 0,Y 98.603,Z 821.567,A -85,B 0,C 180,E1 24389.996,E2 24389.996} C_VEL
LIN {X 0,Y 98.571,Z 817.263,A -85,B 0,C 180,E1 24403.317,E2 24403.317} C_VEL
LIN {X 0,Y 103.265,Z 807.331,A -85,B 0,C 180,E1 24420.871,E2 24420.871} C_VEL
LIN {X 0,Y 116.984,Z 790.022,A -85,B 0,C 180,E1 24438.085,E2 24438.085} C_VEL
LIN {X 0,Y 136.462,Z 767.341,A -85,B 0,C 180,E1 24450.432,E2 24450.432} C_VEL
LIN {X 0,Y 158.43,Z 739.359,A -85,B 0,C 180,E1 24458.921,E2 24458.921} C_VEL
LIN {X 0,Y 177.015,Z 711.58,A -85,B 0,C 180,E1 24464.049,E2 24464.049} C_VEL
LIN {X 0,Y 174.033,Z 690.587,A -85,B 0,C 180,E1 24473.14,E2 24473.14} C_VEL
LIN {X 0,Y 170.111,Z 671.177,A -85,B 0,C 180,E1 24483.042,E2 24483.042} C_VEL
LIN {X 0,Y 166.847,Z 658.137,A -85,B 0,C 180,E1 24491.679,E2 24491.679} C_VEL
LIN {X 0,Y 162.555,Z 649.541,A -85,B 0,C 180,E1 24501.886,E2 24501.886} C_VEL
LIN {X 0,Y 160.792,Z 646.255,A -85,B 0,C 180,E1 24508.099,E2 24508.099} C_VEL
LIN {X 0,Y 158.781,Z 644.932,A -85,B 0,C 180,E1 24520.288,E2 24520.288} C_VEL
LIN {X 0,Y 159.402,Z 646.458,A -85,B 0,C 180,E1 24529.469,E2 24529.469} C_VEL
LIN {X 0,Y 161.283,Z 652.196,A -85,B 0,C 180,E1 24539.762,E2 24539.762} C_VEL
LIN {X 0,Y 164.263,Z 661.624,A -85,B 0,C 180,E1 24549.644,E2 24549.644} C_VEL
LIN {X 0,Y 166.666,Z 672.594,A -85,B 0,C 180,E1 24557.54,E2 24557.54} C_VEL
LIN {X 0,Y 167.542,Z 691.48,A -85,B 0,C 180,E1 24567.412,E2 24567.412} C_VEL
LIN {X 0,Y 167.135,Z 708.078,A -85,B 0,C 180,E1 24575.2,E2 24575.2} C_VEL
LIN {X 0,Y 164.624,Z 712.937,A -85,B 0,C 180,E1 24576.491,E2 24576.491} C_VEL
LIN {X 0,Y 142.419,Z 742.424,A -85,B 0,C 180,E1 24584.603,E2 24584.603} C_VEL
LIN {X 0,Y 127.665,Z 760.086,A -85,B 0,C 180,E1 24592.388,E2 24592.388} C_VEL
LIN {X 0,Y 122.566,Z 764.896,A -85,B 0,C 180,E1 24594.794,E2 24594.794} C_VEL
LIN {X 0,Y 106.532,Z 776.843,A -85,B 0,C 180,E1 24601.709,E2 24601.709} C_VEL
LIN {X 0,Y 105.553,Z 777.876,A -85,B 0,C 180,E1 24602.611,E2 24602.611} C_VEL
LIN {X 0,Y 93.001,Z 794.311,A -85,B 0,C 180,E1 24622.807,E2 24622.807} C_VEL
LIN {X 0,Y 89.01,Z 803.959,A -85,B 0,C 180,E1 24642.661,E2 24642.661} C_VEL
LIN {X 0,Y 93.411,Z 810.836,A -85,B 0,C 180,E1 24664.629,E2 24664.629} C_VEL
LIN {X 0,Y 108.627,Z 814.665,A -85,B 0,C 180,E1 24684.698,E2 24684.698} C_VEL
LIN {X 0,Y 120.547,Z 815.533,A -85,B 0,C 180,E1 24692.911,E2 24692.911} C_VEL
LIN {X 0,Y 114.279,Z 817.123,A -85,B 0,C 180,E1 24697.346,E2 24697.346} C_VEL
LIN {X 0,Y 93.616,Z 821.514,A -85,B 0,C 180,E1 24720.97,E2 24720.97} C_VEL
LIN {X 0,Y 89.852,Z 821.461,A -85,B 0,C 180,E1 24740.295,E2 24740.295} C_VEL
LIN {X 0,Y 90.78,Z 820.212,A -85,B 0,C 180,E1 24749.996,E2 24749.996} C_VEL
LIN {X 0,Y 91.655,Z 813.493,A -85,B 0,C 180,E1 24769.288,E2 24769.288} C_VEL
LIN {X 0,Y 99.832,Z 800.855,A -85,B 0,C 180,E1 24788.915,E2 24788.915} C_VEL
LIN {X 0,Y 116.189,Z 782.435,A -85,B 0,C 180,E1 24804.533,E2 24804.533} C_VEL
LIN {X 0,Y 137.238,Z 758.526,A -85,B 0,C 180,E1 24815.523,E2 24815.523} C_VEL
LIN {X 0,Y 159.788,Z 729.497,A -85,B 0,C 180,E1 24822.959,E2 24822.959} C_VEL
LIN {X 0,Y 170.554,Z 713.722,A -85,B 0,C 180,E1 24825.652,E2 24825.652} C_VEL
LIN {X 0,Y 168.016,Z 693.637,A -85,B 0,C 180,E1 24834.841,E2 24834.841} C_VEL
LIN {X 0,Y 164.955,Z 675.683,A -85,B 0,C 180,E1 24844.563,E2 24844.563} C_VEL
LIN {X 0,Y 162.333,Z 664.021,A -85,B 0,C 180,E1 24852.726,E2 24852.726} C_VEL
LIN {X 0,Y 158.567,Z 656.209,A -85,B 0,C 180,E1 24862.465,E2 24862.465} C_VEL
LIN {X 0,Y 156.718,Z 652.928,A -85,B 0,C 180,E1 24869.605,E2 24869.605} C_VEL
LIN {X 0,Y 155.087,Z 652.195,A -85,B 0,C 180,E1 24883.124,E2 24883.124} C_VEL
LIN {X 0,Y 156.267,Z 655.734,A -85,B 0,C 180,E1 24894.458,E2 24894.458} C_VEL
LIN {X 0,Y 158.383,Z 662.925,A -85,B 0,C 180,E1 24904.3,E2 24904.3} C_VEL
LIN {X 0,Y 161.088,Z 674.475,A -85,B 0,C 180,E1 24914.419,E2 24914.419} C_VEL
LIN {X 0,Y 161.621,Z 689.851,A -85,B 0,C 180,E1 24923.278,E2 24923.278} C_VEL
LIN {X 0,Y 161.058,Z 707.608,A -85,B 0,C 180,E1 24932.225,E2 24932.225} C_VEL
LIN {X 0,Y 160.42,Z 711.817,A -85,B 0,C 180,E1 24934.09,E2 24934.09} C_VEL
LIN {X 0,Y 137.059,Z 742.076,A -85,B 0,C 180,E1 24942.225,E2 24942.225} C_VEL
LIN {X 0,Y 115.881,Z 766.288,A -85,B 0,C 180,E1 24953.816,E2 24953.816} C_VEL
LIN {X 0,Y 105.553,Z 777.876,A -85,B 0,C 180,E1 24962.611,E2 24962.611} C_VEL
LIN {X 0,Y 98.357,Z 783.731,A -85,B 0,C 180,E1 24967.85,E2 24967.85} C_VEL
LIN {X 0,Y 87.335,Z 791.41,A -85,B 0,C 180,E1 24976.945,E2 24976.945} C_VEL
LIN {X 0,Y 86.684,Z 792.221,A -85,B 0,C 180,E1 24978.224,E2 24978.224} C_VEL
LIN {X 0,Y 81.352,Z 802.421,A -85,B 0,C 180,E1 24998.536,E2 24998.536} C_VEL
LIN {X 0,Y 85.414,Z 810.809,A -85,B 0,C 180,E1 25025.063,E2 25025.063} C_VEL
LIN {X 0,Y 101.79,Z 815.447,A -85,B 0,C 180,E1 25046.808,E2 25046.808} C_VEL
LIN {X 0,Y 110.738,Z 816.403,A -85,B 0,C 180,E1 25053.134,E2 25053.134} C_VEL
LIN {X 0,Y 84.553,Z 820.661,A -85,B 0,C 180,E1 25083.5,E2 25083.5} C_VEL
LIN {X 0,Y 82.065,Z 820.083,A -85,B 0,C 180,E1 25099.364,E2 25099.364} C_VEL
LIN {X 0,Y 82.967,Z 818.716,A -85,B 0,C 180,E1 25109.995,E2 25109.995} C_VEL
LIN {X 0,Y 83.618,Z 812.819,A -85,B 0,C 180,E1 25128.469,E2 25128.469} C_VEL
LIN {X 0,Y 91.126,Z 801.383,A -85,B 0,C 180,E1 25148.535,E2 25148.535} C_VEL
LIN {X 0,Y 109.109,Z 782.141,A -85,B 0,C 180,E1 25166.36,E2 25166.36} C_VEL
LIN {X 0,Y 130.99,Z 758.422,A -85,B 0,C 180,E1 25177.614,E2 25177.614} C_VEL
LIN {X 0,Y 154.683,Z 728.947,A -85,B 0,C 180,E1 25185.137,E2 25185.137} C_VEL
LIN {X 0,Y 163.424,Z 716.757,A -85,B 0,C 180,E1 25187.18,E2 25187.18} C_VEL
LIN {X 0,Y 163.356,Z 707.205,A -85,B 0,C 180,E1 25191.349,E2 25191.349} C_VEL
LIN {X 0,Y 160.801,Z 686.781,A -85,B 0,C 180,E1 25202.035,E2 25202.035} C_VEL
LIN {X 0,Y 158.352,Z 671.933,A -85,B 0,C 180,E1 25211.846,E2 25211.846} C_VEL
LIN {X 0,Y 155.074,Z 663.943,A -85,B 0,C 180,E1 25221.181,E2 25221.181} C_VEL
LIN {X 0,Y 152.908,Z 659.852,A -85,B 0,C 180,E1 25229.689,E2 25229.689} C_VEL
LIN {X 0,Y 151.575,Z 658.983,A -85,B 0,C 180,E1 25236.959,E2 25236.959} C_VEL
LIN {X 0,Y 151.389,Z 659.498,A -85,B 0,C 180,E1 25245.57,E2 25245.57} C_VEL
LIN {X 0,Y 152.432,Z 663.461,A -85,B 0,C 180,E1 25255.98,E2 25255.98} C_VEL
LIN {X 0,Y 154.276,Z 671.057,A -85,B 0,C 180,E1 25265.683,E2 25265.683} C_VEL
LIN {X 0,Y 156.096,Z 681.974,A -85,B 0,C 180,E1 25274.943,E2 25274.943} C_VEL
LIN {X 0,Y 155.713,Z 699.714,A -85,B 0,C 180,E1 25285.122,E2 25285.122} C_VEL
LIN {X 0,Y 154.397,Z 713.542,A -85,B 0,C 180,E1 25292.169,E2 25292.169} C_VEL
LIN {X 0,Y 129.879,Z 744.058,A -85,B 0,C 180,E1 25300.534,E2 25300.534} C_VEL
LIN {X 0,Y 107.611,Z 768.301,A -85,B 0,C 180,E1 25312.809,E2 25312.809} C_VEL
LIN {X 0,Y 90.312,Z 787.411,A -85,B 0,C 180,E1 25331.204,E2 25331.204} C_VEL
LIN {X 0,Y 86.684,Z 792.221,A -85,B 0,C 180,E1 25338.224,E2 25338.224} C_VEL
LIN {X 0,Y 81.37,Z 796.724,A -85,B 0,C 180,E1 25345.806,E2 25345.806} C_VEL
LIN {X 0,Y 73.285,Z 803.093,A -85,B 0,C 180,E1 25360.456,E2 25360.456} C_VEL
LIN {X 0,Y 77.572,Z 810.778,A -85,B 0,C 180,E1 25385.948,E2 25385.948} C_VEL
LIN {X 0,Y 100.124,Z 816.742,A -85,B 0,C 180,E1 25412.942,E2 25412.942} C_VEL
LIN {X 0,Y 79.84,Z 819.345,A -85,B 0,C 180,E1 25435.32,E2 25435.32} C_VEL
LIN {X 0,Y 74.306,Z 818.697,A -85,B 0,C 180,E1 25458.238,E2 25458.238} C_VEL
LIN {X 0,Y 75.169,Z 817.205,A -85,B 0,C 180,E1 25469.995,E2 25469.995} C_VEL
LIN {X 0,Y 76.131,Z 810.959,A -85,B 0,C 180,E1 25490.362,E2 25490.362} C_VEL
LIN {X 0,Y 86.667,Z 797.16,A -85,B 0,C 180,E1 25514.324,E2 25514.324} C_VEL
LIN {X 0,Y 107.438,Z 776.501,A -85,B 0,C 180,E1 25531.729,E2 25531.729} C_VEL
LIN {X 0,Y 131.764,Z 750.556,A -85,B 0,C 180,E1 25542.315,E2 25542.315} C_VEL
LIN {X 0,Y 156.393,Z 719.514,A -85,B 0,C 180,E1 25548.926,E2 25548.926} C_VEL
LIN {X 0,Y 157.591,Z 716.867,A -85,B 0,C 180,E1 25549.634,E2 25549.634} C_VEL
LIN {X 0,Y 155.945,Z 697.07,A -85,B 0,C 180,E1 25560.012,E2 25560.012} C_VEL
LIN {X 0,Y 154.16,Z 681.244,A -85,B 0,C 180,E1 25570.053,E2 25570.053} C_VEL
LIN {X 0,Y 152.619,Z 674.823,A -85,B 0,C 180,E1 25575.836,E2 25575.836} C_VEL
LIN {X 0,Y 149.988,Z 668.813,A -85,B 0,C 180,E1 25584.705,E2 25584.705} C_VEL
LIN {X 0,Y 148.67,Z 666.584,A -85,B 0,C 180,E1 25590.624,E2 25590.624} C_VEL
LIN {X 0,Y 147.276,Z 666.132,A -85,B 0,C 180,E1 25603.98,E2 25603.98} C_VEL
LIN {X 0,Y 148.086,Z 669.684,A -85,B 0,C 180,E1 25614.898,E2 25614.898} C_VEL
LIN {X 0,Y 149.314,Z 675.778,A -85,B 0,C 180,E1 25623.521,E2 25623.521} C_VEL
LIN {X 0,Y 150.87,Z 686.242,A -85,B 0,C 180,E1 25633.214,E2 25633.214} C_VEL
LIN {X 0,Y 149.928,Z 702.679,A -85,B 0,C 180,E1 25643.27,E2 25643.27} C_VEL
LIN {X 0,Y 147.988,Z 715.888,A -85,B 0,C 180,E1 25650.24,E2 25650.24} C_VEL
LIN {X 0,Y 122.573,Z 746.138,A -85,B 0,C 180,E1 25658.726,E2 25658.726} C_VEL
LIN {X 0,Y 99.719,Z 769.842,A -85,B 0,C 180,E1 25671.311,E2 25671.311} C_VEL
LIN {X 0,Y 82.579,Z 787.871,A -85,B 0,C 180,E1 25689.992,E2 25689.992} C_VEL
LIN {X 0,Y 74.819,Z 798.762,A -85,B 0,C 180,E1 25709.581,E2 25709.581} C_VEL
LIN {X 0,Y 73.285,Z 803.093,A -85,B 0,C 180,E1 25720.456,E2 25720.456} C_VEL
LIN {X 0,Y 71.059,Z 806.415,A -85,B 0,C 180,E1 25730.389,E2 25730.389} C_VEL
LIN {X 0,Y 70.138,Z 810.83,A -85,B 0,C 180,E1 25748.037,E2 25748.037} C_VEL
LIN {X 0,Y 89.15,Z 816.569,A -85,B 0,C 180,E1 25772.45,E2 25772.45} C_VEL
LIN {X 0,Y 84.954,Z 817.278,A -85,B 0,C 180,E1 25777.137,E2 25777.137} C_VEL
LIN {X 0,Y 68.507,Z 818.046,A -85,B 0,C 180,E1 25803.761,E2 25803.761} C_VEL
LIN {X 0,Y 67.366,Z 815.666,A -85,B 0,C 180,E1 25829.994,E2 25829.994} C_VEL
LIN {X 0,Y 68.676,Z 809.051,A -85,B 0,C 180,E1 25852.688,E2 25852.688} C_VEL
LIN {X 0,Y 81.034,Z 794.66,A -85,B 0,C 180,E1 25878.356,E2 25878.356} C_VEL
LIN {X 0,Y 103.776,Z 773.277,A -85,B 0,C 180,E1 25895.755,E2 25895.755} C_VEL
LIN {X 0,Y 129.307,Z 746.712,A -85,B 0,C 180,E1 25905.765,E2 25905.765} C_VEL
LIN {X 0,Y 151.236,Z 719.394,A -85,B 0,C 180,E1 25911.323,E2 25911.323} C_VEL
LIN {X 0,Y 150.335,Z 701.657,A -85,B 0,C 180,E1 25921.207,E2 25921.207} C_VEL
LIN {X 0,Y 149.11,Z 685.853,A -85,B 0,C 180,E1 25931.729,E2 25931.729} C_VEL
LIN {X 0,Y 147.115,Z 678.554,A -85,B 0,C 180,E1 25939.555,E2 25939.555} C_VEL
LIN {X 0,Y 144.777,Z 673.702,A -85,B 0,C 180,E1 25949.472,E2 25949.472} C_VEL
LIN {X 0,Y 143.079,Z 672.787,A -85,B 0,C 180,E1 25962.209,E2 25962.209} C_VEL
LIN {X 0,Y 143.624,Z 675.769,A -85,B 0,C 180,E1 25973.637,E2 25973.637} C_VEL
LIN {X 0,Y 144.675,Z 682.917,A -85,B 0,C 180,E1 25984.081,E2 25984.081} C_VEL
LIN {X 0,Y 145.474,Z 692.77,A -85,B 0,C 180,E1 25993.171,E2 25993.171} C_VEL
LIN {X 0,Y 143.742,Z 708.892,A -85,B 0,C 180,E1 26003.197,E2 26003.197} C_VEL
LIN {X 0,Y 142.606,Z 716.329,A -85,B 0,C 180,E1 26007.489,E2 26007.489} C_VEL
LIN {X 0,Y 131.717,Z 730.19,A -85,B 0,C 180,E1 26010.956,E2 26010.956} C_VEL
LIN {X 0,Y 106.057,Z 757.649,A -85,B 0,C 180,E1 26020.885,E2 26020.885} C_VEL
LIN {X 0,Y 83.17,Z 779.781,A -85,B 0,C 180,E1 26037.401,E2 26037.401} C_VEL
LIN {X 0,Y 69.793,Z 794.412,A -85,B 0,C 180,E1 26059.364,E2 26059.364} C_VEL
LIN {X 0,Y 65.322,Z 804.943,A -85,B 0,C 180,E1 26086.57,E2 26086.57} C_VEL
LIN {X 0,Y 70.138,Z 810.83,A -85,B 0,C 180,E1 26108.037,E2 26108.037} C_VEL
LIN {X 0,Y 70.699,Z 812.832,A -85,B 0,C 180,E1 26117.497,E2 26117.497} C_VEL
LIN {X 0,Y 72.953,Z 814.659,A -85,B 0,C 180,E1 26126.696,E2 26126.696} C_VEL
LIN {X 0,Y 79.207,Z 816.146,A -85,B 0,C 180,E1 26132.802,E2 26132.802} C_VEL
LIN {X 0,Y 61.441,Z 816.575,A -85,B 0,C 180,E1 26160.465,E2 26160.465} C_VEL
LIN {X 0,Y 59.596,Z 813.953,A -85,B 0,C 180,E1 26189.994,E2 26189.994} C_VEL
LIN {X 0,Y 61.378,Z 806.909,A -85,B 0,C 180,E1 26215.568,E2 26215.568} C_VEL
LIN {X 0,Y 74.722,Z 793.001,A -85,B 0,C 180,E1 26241.729,E2 26241.729} C_VEL
LIN {X 0,Y 97.589,Z 772.719,A -85,B 0,C 180,E1 26258.563,E2 26258.563} C_VEL
LIN {X 0,Y 123.671,Z 746.764,A -85,B 0,C 180,E1 26268.339,E2 26268.339} C_VEL
LIN {X 0,Y 144.978,Z 721.228,A -85,B 0,C 180,E1 26273.558,E2 26273.558} C_VEL
LIN {X 0,Y 144.549,Z 702.821,A -85,B 0,C 180,E1 26284.518,E2 26284.518} C_VEL
LIN {X 0,Y 143.959,Z 690.266,A -85,B 0,C 180,E1 26293.666,E2 26293.666} C_VEL
LIN {X 0,Y 141.986,Z 683.46,A -85,B 0,C 180,E1 26302.343,E2 26302.343} C_VEL
LIN {X 0,Y 139.778,Z 679.718,A -85,B 0,C 180,E1 26312.807,E2 26312.807} C_VEL
LIN {X 0,Y 138.838,Z 679.385,A -85,B 0,C 180,E1 26320.884,E2 26320.884} C_VEL
LIN {X 0,Y 139.147,Z 682.085,A -85,B 0,C 180,E1 26332.881,E2 26332.881} C_VEL
LIN {X 0,Y 139.822,Z 688.917,A -85,B 0,C 180,E1 26343.411,E2 26343.411} C_VEL
LIN {X 0,Y 140.167,Z 696.609,A -85,B 0,C 180,E1 26351.094,E2 26351.094} C_VEL
LIN {X 0,Y 138.05,Z 711.182,A -85,B 0,C 180,E1 26360.852,E2 26360.852} C_VEL
LIN {X 0,Y 136.1,Z 719.663,A -85,B 0,C 180,E1 26365.754,E2 26365.754} C_VEL
LIN {X 0,Y 109.256,Z 749.178,A -85,B 0,C 180,E1 26374.043,E2 26374.043} C_VEL
LIN {X 0,Y 82.876,Z 773.967,A -85,B 0,C 180,E1 26388.589,E2 26388.589} C_VEL
LIN {X 0,Y 64.973,Z 790.983,A -85,B 0,C 180,E1 26410.841,E2 26410.841} C_VEL
LIN {X 0,Y 58.004,Z 800.773,A -85,B 0,C 180,E1 26434.251,E2 26434.251} C_VEL
LIN {X 0,Y 60.855,Z 809.558,A -85,B 0,C 180,E1 26465.559,E2 26465.559} C_VEL
LIN {X 0,Y 72.953,Z 814.659,A -85,B 0,C 180,E1 26486.696,E2 26486.696} C_VEL
LIN {X 0,Y 72.629,Z 815.396,A -85,B 0,C 180,E1 26491.1,E2 26491.1} C_VEL
LIN {X 0,Y 64.789,Z 815.59,A -85,B 0,C 180,E1 26498.886,E2 26498.886} C_VEL
LIN {X 0,Y 60.337,Z 815.441,A -85,B 0,C 180,E1 26504.066,E2 26504.066} C_VEL
LIN {X 0,Y 51.294,Z 814.021,A -85,B 0,C 180,E1 26532.824,E2 26532.824} C_VEL
LIN {X 0,Y 51.833,Z 812.185,A -85,B 0,C 180,E1 26549.993,E2 26549.993} C_VEL
LIN {X 0,Y 54.259,Z 804.761,A -85,B 0,C 180,E1 26579.223,E2 26579.223} C_VEL
LIN {X 0,Y 71.256,Z 789.176,A -85,B 0,C 180,E1 26608.194,E2 26608.194} C_VEL
LIN {X 0,Y 96.424,Z 767.931,A -85,B 0,C 180,E1 26623.885,E2 26623.885} C_VEL
LIN {X 0,Y 124.31,Z 740.3,A -85,B 0,C 180,E1 26632.643,E2 26632.643} C_VEL
LIN {X 0,Y 138.739,Z 722.953,A -85,B 0,C 180,E1 26635.95,E2 26635.95} C_VEL
LIN {X 0,Y 138.988,Z 705.508,A -85,B 0,C 180,E1 26647.131,E2 26647.131} C_VEL
LIN {X 0,Y 138.822,Z 695.123,A -85,B 0,C 180,E1 26655.405,E2 26655.405} C_VEL
LIN {X 0,Y 137.071,Z 689.231,A -85,B 0,C 180,E1 26663.872,E2 26663.872} C_VEL
LIN {X 0,Y 135.082,Z 686.229,A -85,B 0,C 180,E1 26674.1,E2 26674.1} C_VEL
LIN {X 0,Y 134.203,Z 686.998,A -85,B 0,C 180,E1 26687.401,E2 26687.401} C_VEL
LIN {X 0,Y 134.664,Z 690.021,A -85,B 0,C 180,E1 26695.798,E2 26695.798} C_VEL
LIN {X 0,Y 134.838,Z 697.024,A -85,B 0,C 180,E1 26705.319,E2 26705.319} C_VEL
LIN {X 0,Y 134.339,Z 704.294,A -85,B 0,C 180,E1 26711.947,E2 26711.947} C_VEL
LIN {X 0,Y 131.393,Z 718.475,A -85,B 0,C 180,E1 26721.513,E2 26721.513} C_VEL
LIN {X 0,Y 130.093,Z 721.821,A -85,B 0,C 180,E1 26723.319,E2 26723.319} C_VEL
LIN {X 0,Y 101.617,Z 751.816,A -85,B 0,C 180,E1 26731.691,E2 26731.691} C_VEL
LIN {X 0,Y 74.522,Z 775.774,A -85,B 0,C 180,E1 26746.751,E2 26746.751} C_VEL
LIN {X 0,Y 56.218,Z 792.305,A -85,B 0,C 180,E1 26771.158,E2 26771.158} C_VEL
LIN {X 0,Y 49.51,Z 802.903,A -85,B 0,C 180,E1 26802.155,E2 26802.155} C_VEL
LIN {X 0,Y 60.124,Z 812.595,A -85,B 0,C 180,E1 26842.16,E2 26842.16} C_VEL
LIN {X 0,Y 69.006,Z 815.281,A -85,B 0,C 180,E1 26852.969,E2 26852.969} C_VEL
LIN {X 0,Y 60.337,Z 815.441,A -85,B 0,C 180,E1 26864.066,E2 26864.066} C_VEL
LIN {X 0,Y 52.5,Z 814.596,A -85,B 0,C 180,E1 26874.696,E2 26874.696} C_VEL
LIN {X 0,Y 43.256,Z 811.502,A -85,B 0,C 180,E1 26898.611,E2 26898.611} C_VEL
LIN {X 0,Y 44.056,Z 810.392,A -85,B 0,C 180,E1 26909.991,E2 26909.991} C_VEL
LIN {X 0,Y 47.45,Z 802.514,A -85,B 0,C 180,E1 26943.936,E2 26943.936} C_VEL
LIN {X 0,Y 67.292,Z 786.296,A -85,B 0,C 180,E1 26974.145,E2 26974.145} C_VEL
LIN {X 0,Y 95.466,Z 763.362,A -85,B 0,C 180,E1 26989.025,E2 26989.025} C_VEL
LIN {X 0,Y 123.522,Z 735.71,A -85,B 0,C 180,E1 26996.466,E2 26996.466} C_VEL
LIN {X 0,Y 132.618,Z 724.971,A -85,B 0,C 180,E1 26998.378,E2 26998.378} C_VEL
LIN {X 0,Y 133.522,Z 709.15,A -85,B 0,C 180,E1 27009.23,E2 27009.23} C_VEL
LIN {X 0,Y 133.679,Z 700.596,A -85,B 0,C 180,E1 27016.462,E2 27016.462} C_VEL
LIN {X 0,Y 132.428,Z 695.713,A -85,B 0,C 180,E1 27023.851,E2 27023.851} C_VEL
LIN {X 0,Y 130.303,Z 692.636,A -85,B 0,C 180,E1 27035.579,E2 27035.579} C_VEL
LIN {X 0,Y 129.593,Z 693.18,A -85,B 0,C 180,E1 27045.497,E2 27045.497} C_VEL
LIN {X 0,Y 129.776,Z 695.92,A -85,B 0,C 180,E1 27054.775,E2 27054.775} C_VEL
LIN {X 0,Y 129.629,Z 702.423,A -85,B 0,C 180,E1 27064.256,E2 27064.256} C_VEL
LIN {X 0,Y 128.789,Z 709.404,A -85,B 0,C 180,E1 27070.837,E2 27070.837} C_VEL
LIN {X 0,Y 125.421,Z 722.154,A -85,B 0,C 180,E1 27079.908,E2 27079.908} C_VEL
LIN {X 0,Y 122.668,Z 725.861,A -85,B 0,C 180,E1 27080.989,E2 27080.989} C_VEL
LIN {X 0,Y 92.749,Z 755.462,A -85,B 0,C 180,E1 27089.545,E2 27089.545} C_VEL
LIN {X 0,Y 65.785,Z 777.911,A -85,B 0,C 180,E1 27104.858,E2 27104.858} C_VEL
LIN {X 0,Y 46.866,Z 794.097,A -85,B 0,C 180,E1 27133.124,E2 27133.124} C_VEL
LIN {X 0,Y 42.257,Z 805.234,A -85,B 0,C 180,E1 27174.818,E2 27174.818} C_VEL
LIN {X 0,Y 58.308,Z 813.878,A -85,B 0,C 180,E1 27212.759,E2 27212.759} C_VEL
LIN {X 0,Y 48.2,Z 813.49,A -85,B 0,C 180,E1 27231.069,E2 27231.069} C_VEL
LIN {X 0,Y 43.256,Z 811.502,A -85,B 0,C 180,E1 27258.611,E2 27258.611} C_VEL
LIN {X 0,Y 41.512,Z 809.333,A -85,B 0,C 180,E1 27272.773,E2 27272.773} C_VEL
LIN {X 0,Y 39.904,Z 801.156,A -85,B 0,C 180,E1 27306.569,E2 27306.569} C_VEL
LIN {X 0,Y 61.961,Z 784.756,A -85,B 0,C 180,E1 27339.149,E2 27339.149} C_VEL
LIN {X 0,Y 89.941,Z 763.236,A -85,B 0,C 180,E1 27352.64,E2 27352.64} C_VEL
LIN {X 0,Y 119.229,Z 735.286,A -85,B 0,C 180,E1 27359.608,E2 27359.608} C_VEL
LIN {X 0,Y 126.593,Z 726.829,A -85,B 0,C 180,E1 27361.071,E2 27361.071} C_VEL
LIN {X 0,Y 128.044,Z 712.133,A -85,B 0,C 180,E1 27371.957,E2 27371.957} C_VEL
LIN {X 0,Y 128.223,Z 704.834,A -85,B 0,C 180,E1 27379.162,E2 27379.162} C_VEL
LIN {X 0,Y 126.638,Z 700.278,A -85,B 0,C 180,E1 27388.586,E2 27388.586} C_VEL
LIN {X 0,Y 125.257,Z 699.092,A -85,B 0,C 180,E1 27397.202,E2 27397.202} C_VEL
LIN {X 0,Y 124.756,Z 699.777,A -85,B 0,C 180,E1 27406.753,E2 27406.753} C_VEL
LIN {X 0,Y 124.725,Z 703.528,A -85,B 0,C 180,E1 27417.127,E2 27417.127} C_VEL
LIN {X 0,Y 124.031,Z 710.805,A -85,B 0,C 180,E1 27426.629,E2 27426.629} C_VEL
LIN {X 0,Y 120.147,Z 723.705,A -85,B 0,C 180,E1 27436.724,E2 27436.724} C_VEL
LIN {X 0,Y 118.182,Z 726.618,A -85,B 0,C 180,E1 27437.833,E2 27437.833} C_VEL
LIN {X 0,Y 87.442,Z 756.145,A -85,B 0,C 180,E1 27445.71,E2 27445.71} C_VEL
LIN {X 0,Y 58.981,Z 778.542,A -85,B 0,C 180,E1 27460.761,E2 27460.761} C_VEL
LIN {X 0,Y 39.378,Z 793.872,A -85,B 0,C 180,E1 27489.666,E2 27489.666} C_VEL
LIN {X 0,Y 34.917,Z 805.192,A -85,B 0,C 180,E1 27539.948,E2 27539.948} C_VEL
LIN {X 0,Y 47.519,Z 811.989,A -85,B 0,C 180,E1 27572.391,E2 27572.391} C_VEL
LIN {X 0,Y 40.984,Z 811.592,A -85,B 0,C 180,E1 27587.566,E2 27587.566} C_VEL
LIN {X 0,Y 36.325,Z 808.405,A -85,B 0,C 180,E1 27629.99,E2 27629.99} C_VEL
LIN {X 0,Y 39.904,Z 801.156,A -85,B 0,C 180,E1 27666.569,E2 27666.569} C_VEL
LIN {X 0,Y 43.574,Z 795.915,A -85,B 0,C 180,E1 27682.324,E2 27682.324} C_VEL
LIN {X 0,Y 51.999,Z 786.69,A -85,B 0,C 180,E1 27701.123,E2 27701.123} C_VEL
LIN {X 0,Y 53.525,Z 785.64,A -85,B 0,C 180,E1 27702.435,E2 27702.435} C_VEL
LIN {X 0,Y 83.442,Z 764.119,A -85,B 0,C 180,E1 27716.291,E2 27716.291} C_VEL
LIN {X 0,Y 113.342,Z 736.952,A -85,B 0,C 180,E1 27722.658,E2 27722.658} C_VEL
LIN {X 0,Y 120.099,Z 729.829,A -85,B 0,C 180,E1 27723.667,E2 27723.667} C_VEL
LIN {X 0,Y 121.579,Z 723.304,A -85,B 0,C 180,E1 27728.069,E2 27728.069} C_VEL
LIN {X 0,Y 123.056,Z 712.768,A -85,B 0,C 180,E1 27737.108,E2 27737.108} C_VEL
LIN {X 0,Y 122.582,Z 708.254,A -85,B 0,C 180,E1 27743.813,E2 27743.813} C_VEL
LIN {X 0,Y 121.523,Z 706.295,A -85,B 0,C 180,E1 27749.908,E2 27749.908} C_VEL
LIN {X 0,Y 119.994,Z 705.461,A -85,B 0,C 180,E1 27760.798,E2 27760.798} C_VEL
LIN {X 0,Y 119.774,Z 707.478,A -85,B 0,C 180,E1 27772.471,E2 27772.471} C_VEL
LIN {X 0,Y 119.063,Z 712.769,A -85,B 0,C 180,E1 27781.605,E2 27781.605} C_VEL
LIN {X 0,Y 117.461,Z 719.096,A -85,B 0,C 180,E1 27788.252,E2 27788.252} C_VEL
LIN {X 0,Y 114.703,Z 726.583,A -85,B 0,C 180,E1 27794.205,E2 27794.205} C_VEL
LIN {X 0,Y 84.548,Z 755.055,A -85,B 0,C 180,E1 27800.824,E2 27800.824} C_VEL
LIN {X 0,Y 53.308,Z 778.613,A -85,B 0,C 180,E1 27815.058,E2 27815.058} C_VEL
LIN {X 0,Y 32.162,Z 793.484,A -85,B 0,C 180,E1 27844.431,E2 27844.431} C_VEL
LIN {X 0,Y 28.009,Z 805.095,A -85,B 0,C 180,E1 27907.701,E2 27907.701} C_VEL
LIN {X 0,Y 33.847,Z 808.398,A -85,B 0,C 180,E1 27926.511,E2 27926.511} C_VEL
LIN {X 0,Y 37.187,Z 809.998,A -85,B 0,C 180,E1 27935.464,E2 27935.464} C_VEL
LIN {X 0,Y 28.573,Z 806.359,A -85,B 0,C 180,E1 27989.987,E2 27989.987} C_VEL
LIN {X 0,Y 35.159,Z 797.674,A -85,B 0,C 180,E1 28038.157,E2 28038.157} C_VEL
LIN {X 0,Y 53.525,Z 785.64,A -85,B 0,C 180,E1 28062.435,E2 28062.435} C_VEL
LIN {X 0,Y 59.117,Z 781.207,A -85,B 0,C 180,E1 28067.603,E2 28067.603} C_VEL
LIN {X 0,Y 73.738,Z 767.54,A -85,B 0,C 180,E1 28079.565,E2 28079.565} C_VEL
LIN {X 0,Y 75.42,Z 766.252,A -85,B 0,C 180,E1 28080.066,E2 28080.066} C_VEL
LIN {X 0,Y 107.598,Z 738.555,A -85,B 0,C 180,E1 28085.998,E2 28085.998} C_VEL
LIN {X 0,Y 115.11,Z 730.699,A -85,B 0,C 180,E1 28087.069,E2 28087.069} C_VEL
LIN {X 0,Y 117.387,Z 719.344,A -85,B 0,C 180,E1 28096.886,E2 28096.886} C_VEL
LIN {X 0,Y 117.556,Z 714.902,A -85,B 0,C 180,E1 28102.746,E2 28102.746} C_VEL
LIN {X 0,Y 116.04,Z 712.247,A -85,B 0,C 180,E1 28111.478,E2 28111.478} C_VEL
LIN {X 0,Y 114.911,Z 711.656,A -85,B 0,C 180,E1 28121.228,E2 28121.228} C_VEL
LIN {X 0,Y 114.605,Z 713.6,A -85,B 0,C 180,E1 28132.459,E2 28132.459} C_VEL
LIN {X 0,Y 113.461,Z 718.936,A -85,B 0,C 180,E1 28141.708,E2 28141.708} C_VEL
LIN {X 0,Y 111.126,Z 725.185,A -85,B 0,C 180,E1 28147.999,E2 28147.999} C_VEL
LIN {X 0,Y 109.484,Z 728.857,A -85,B 0,C 180,E1 28150.931,E2 28150.931} C_VEL
LIN {X 0,Y 77.819,Z 757.467,A -85,B 0,C 180,E1 28156.704,E2 28156.704} C_VEL
LIN {X 0,Y 45.453,Z 780.38,A -85,B 0,C 180,E1 28170.008,E2 28170.008} C_VEL
LIN {X 0,Y 22.841,Z 794.764,A -85,B 0,C 180,E1 28203.907,E2 28203.907} C_VEL
LIN {X 0,Y 24.233,Z 806.044,A -85,B 0,C 180,E1 28287.858,E2 28287.858} C_VEL
LIN {X 0,Y 26.909,Z 807.152,A -85,B 0,C 180,E1 28294.157,E2 28294.157} C_VEL
LIN {X 0,Y 20.837,Z 804.26,A -85,B 0,C 180,E1 28349.982,E2 28349.982} C_VEL
LIN {X 0,Y 30.104,Z 795.248,A -85,B 0,C 180,E1 28408.921,E2 28408.921} C_VEL
LIN {X 0,Y 59.226,Z 777.662,A -85,B 0,C 180,E1 28434.699,E2 28434.699} C_VEL
LIN {X 0,Y 75.42,Z 766.252,A -85,B 0,C 180,E1 28440.066,E2 28440.066} C_VEL
LIN {X 0,Y 81.612,Z 760.981,A -85,B 0,C 180,E1 28442.396,E2 28442.396} C_VEL
LIN {X 0,Y 96.822,Z 745.108,A -85,B 0,C 180,E1 28449.034,E2 28449.034} C_VEL
LIN {X 0,Y 98.394,Z 743.595,A -85,B 0,C 180,E1 28449.267,E2 28449.267} C_VEL
LIN {X 0,Y 109.752,Z 732.209,A -85,B 0,C 180,E1 28450.849,E2 28450.849} C_VEL
LIN {X 0,Y 112.126,Z 722.877,A -85,B 0,C 180,E1 28459.742,E2 28459.742} C_VEL
LIN {X 0,Y 111.646,Z 719.346,A -85,B 0,C 180,E1 28466.642,E2 28466.642} C_VEL
LIN {X 0,Y 110.308,Z 717.966,A -85,B 0,C 180,E1 28474.565,E2 28474.565} C_VEL
LIN {X 0,Y 109.332,Z 718.306,A -85,B 0,C 180,E1 28486.183,E2 28486.183} C_VEL
LIN {X 0,Y 109.094,Z 720.127,A -85,B 0,C 180,E1 28493.604,E2 28493.604} C_VEL
LIN {X 0,Y 107.393,Z 725.576,A -85,B 0,C 180,E1 28502.485,E2 28502.485} C_VEL
LIN {X 0,Y 105.035,Z 730.441,A -85,B 0,C 180,E1 28506.919,E2 28506.919} C_VEL
LIN {X 0,Y 74.754,Z 757.264,A -85,B 0,C 180,E1 28511.23,E2 28511.23} C_VEL
LIN {X 0,Y 42.067,Z 779.708,A -85,B 0,C 180,E1 28520.715,E2 28520.715} C_VEL
LIN {X 0,Y 16.239,Z 794.227,A -85,B 0,C 180,E1 28550.884,E2 28550.884} C_VEL
LIN {X 0,Y 15.938,Z 803.783,A -85,B 0,C 180,E1 28655.751,E2 28655.751} C_VEL
LIN {X 0,Y 13.887,Z 803.334,A -85,B 0,C 180,E1 28676.934,E2 28676.934} C_VEL
LIN {X 0,Y 13.138,Z 801.957,A -85,B 0,C 180,E1 28709.971,E2 28709.971} C_VEL
LIN {X 0,Y 28.318,Z 791.682,A -85,B 0,C 180,E1 28785.434,E2 28785.434} C_VEL
LIN {X 0,Y 57.812,Z 774.895,A -85,B 0,C 180,E1 28802.212,E2 28802.212} C_VEL
LIN {X 0,Y 89.893,Z 751.046,A -85,B 0,C 180,E1 28808.328,E2 28808.328} C_VEL
LIN {X 0,Y 98.394,Z 743.595,A -85,B 0,C 180,E1 28809.267,E2 28809.267} C_VEL
LIN {X 0,Y 102.936,Z 737.781,A -85,B 0,C 180,E1 28811.777,E2 28811.777} C_VEL
LIN {X 0,Y 105.994,Z 729.632,A -85,B 0,C 180,E1 28819.137,E2 28819.137} C_VEL
LIN {X 0,Y 106.5,Z 725.662,A -85,B 0,C 180,E1 28825.264,E2 28825.264} C_VEL
LIN {X 0,Y 104.898,Z 723.876,A -85,B 0,C 180,E1 28835.284,E2 28835.284} C_VEL
LIN {X 0,Y 103.991,Z 724.28,A -85,B 0,C 180,E1 28846.741,E2 28846.741} C_VEL
LIN {X 0,Y 103.025,Z 727.377,A -85,B 0,C 180,E1 28856.286,E2 28856.286} C_VEL
LIN {X 0,Y 101.171,Z 731.479,A -85,B 0,C 180,E1 28861.989,E2 28861.989} C_VEL
LIN {X 0,Y 100.411,Z 732.686,A -85,B 0,C 180,E1 28863.109,E2 28863.109} C_VEL
LIN {X 0,Y 67.875,Z 760.411,A -85,B 0,C 180,E1 28865.834,E2 28865.834} C_VEL
LIN {X 0,Y 34.611,Z 781.937,A -85,B 0,C 180,E1 28871.452,E2 28871.452} C_VEL
LIN {X 0,Y 8.032,Z 795.102,A -85,B 0,C 180,E1 28890.047,E2 28890.047} C_VEL
LIN {X 0,Y 5.832,Z 800.214,A -85,B 0,C 180,E1 29030.663,E2 29030.663} C_VEL
LIN {X 0,Y 6.207,Z 798.446,A -85,B 0,C 180,E1 29107.498,E2 29107.498} C_VEL
LIN {X 0,Y 34.175,Z 785.401,A -85,B 0,C 180,E1 29164.713,E2 29164.713} C_VEL
LIN {X 0,Y 67.497,Z 765.322,A -85,B 0,C 180,E1 29171.291,E2 29171.291} C_VEL
LIN {X 0,Y 100.185,Z 738.616,A -85,B 0,C 180,E1 29173.936,E2 29173.936} C_VEL
LIN {X 0,Y 104.446,Z 734.395,A -85,B 0,C 180,E1 29174.323,E2 29174.323} C_VEL
LIN {X 0,Y 105.994,Z 729.632,A -85,B 0,C 180,E1 29179.137,E2 29179.137} C_VEL
LIN {X 0,Y 105.394,Z 727.424,A -85,B 0,C 180,E1 29184.17,E2 29184.17} C_VEL
LIN {X 0,Y 98.914,Z 729.636,A -85,B 0,C 180,E1 29198.673,E2 29198.673} C_VEL
LIN {X 0,Y 97.739,Z 731.964,A -85,B 0,C 180,E1 29213.783,E2 29213.783} C_VEL
LIN {X 0,Y 96.579,Z 734.289,A -85,B 0,C 180,E1 29217.955,E2 29217.955} C_VEL
LIN {X 0,Y 91.756,Z 739.105,A -85,B 0,C 180,E1 29218.811,E2 29218.811} C_VEL
LIN {X 0,Y 57.611,Z 766.291,A -85,B 0,C 180,E1 29219.23,E2 29219.23} C_VEL
LIN {X 0,Y 23.486,Z 786.751,A -85,B 0,C 180,E1 29216.162,E2 29216.162} C_VEL
LIN {X 0,Y 8.948,Z 793.986,A -85,B 0,C 180,E1 29195.584,E2 29195.584} C_VEL
LIN {X 0,Y 10.523,Z 793.65,A -85,B 0,C 180,E1 29182.986,E2 29182.986} C_VEL
LIN {X 0,Y 45.676,Z 776.741,A -85,B 0,C 180,E1 29177.662,E2 29177.662} C_VEL
LIN {X 0,Y 79.619,Z 753.676,A -85,B 0,C 180,E1 29178.06,E2 29178.06} C_VEL
LIN {X 0,Y 99.413,Z 736.57,A -85,B 0,C 180,E1 29178.337,E2 29178.337} C_VEL
LIN {X 0,Y 100.774,Z 733.005,A -85,B 0,C 180,E1 29182.172,E2 29182.172} C_VEL
LIN {X 0,Y 100.617,Z 730.964,A -85,B 0,C 180,E1 29186.855,E2 29186.855} C_VEL
LIN {X 0,Y 98.914,Z 729.636,A -85,B 0,C 180,E1 29198.673,E2 29198.673} C_VEL
LIN {X 0,Y 96.785,Z 731.602,A -85,B 0,C 180,E1 29203.488,E2 29203.488} C_VEL
LIN {X 0,Y 92.125,Z 736.887,A -85,B 0,C 180,E1 29211.616,E2 29211.616} C_VEL
LIN {X 0,Y 91.842,Z 737.484,A -85,B 0,C 180,E1 29213.348,E2 29213.348} C_VEL
LIN {X 0,Y 85.972,Z 742.965,A -85,B 0,C 180,E1 29213.738,E2 29213.738} C_VEL
LIN {X 0,Y 53.445,Z 768.311,A -85,B 0,C 180,E1 29210.754,E2 29210.754} C_VEL
LIN {X 0,Y 24.84,Z 786.075,A -85,B 0,C 180,E1 29197.646,E2 29197.646} C_VEL
LIN {X 0,Y 50.668,Z 771.869,A -85,B 0,C 180,E1 29186.319,E2 29186.319} C_VEL
LIN {X 0,Y 82.477,Z 749.072,A -85,B 0,C 180,E1 29183.395,E2 29183.395} C_VEL
LIN {X 0,Y 93.416,Z 739.622,A -85,B 0,C 180,E1 29182.913,E2 29182.913} C_VEL
LIN {X 0,Y 94.97,Z 737.88,A -85,B 0,C 180,E1 29183.607,E2 29183.607} C_VEL
LIN {X 0,Y 94.54,Z 736.351,A -85,B 0,C 180,E1 29188.736,E2 29188.736} C_VEL
LIN {X 0,Y 93.051,Z 735.382,A -85,B 0,C 180,E1 29200.631,E2 29200.631} C_VEL
LIN {X 0,Y 92.125,Z 736.887,A -85,B 0,C 180,E1 29211.616,E2 29211.616} C_VEL
LIN {X 0,Y 89.422,Z 739.665,A -85,B 0,C 180,E1 29212.726,E2 29212.726} C_VEL
LIN {X 0,Y 74.924,Z 751.794,A -85,B 0,C 180,E1 29207.062,E2 29207.062} C_VEL
LIN {X 0,Y 46.157,Z 773.374,A -85,B 0,C 180,E1 29199.164,E2 29199.164} C_VEL
LIN {X 0,Y 47.837,Z 772.429,A -85,B 0,C 180,E1 29196.262,E2 29196.262} C_VEL
LIN {X 0,Y 78.716,Z 750.446,A -85,B 0,C 180,E1 29189.23,E2 29189.23} C_VEL
LIN {X 0,Y 88.766,Z 741.918,A -85,B 0,C 180,E1 29188.266,E2 29188.266} C_VEL
LIN {X 0,Y 86.547,Z 741.689,A -85,B 0,C 180,E1 29207.561,E2 29207.561} C_VEL
LIN {X 0,Y 83.516,Z 744.425,A -85,B 0,C 180,E1 29208.219,E2 29208.219} C_VEL
LIN {X 0,Y 74.924,Z 751.794,A -85,B 0,C 180,E1 29207.062,E2 29207.062} C_VEL
LIN {X 0,Y 73.604,Z 752.834,A -85,B 0,C 180,E1 29204.593,E2 29204.593} C_VEL
LIN {X 0,Y 77.666,Z 749.93,A -85,B 0,C 180,E1 29196.779,E2 29196.779} C_VEL
LIN {X 0,Y 81.248,Z 747.056,A -85,B 0,C 180,E1 29194.645,E2 29194.645} C_VEL
LIN {X 0,Y 81.52,Z 746.775,A -85,B 0,C 180,E1 29194.878,E2 29194.878} C_VEL
LIN {X 0,Y 80.855,Z 746.665,A -85,B 0,C 180,E1 29201.501,E2 29201.501} C_VEL
LIN {X 0,Y 73.477,Z 753.074,A -85,B 0,C 180,E1 29200.561,E2 29200.561} C_VEL
LIN {X 0,Y 67.292,Z 758.228,A -85,B 0,C 180,E1 29198.825,E2 29198.825} C_VEL
LIN {X 0,Y 71.541,Z 754.996,A -85,B 0,C 180,E1 29196.563,E2 29196.563} C_VEL
LIN {X 0,Y 81.52,Z 746.775,A -85,B 0,C 180,E1 29194.878,E2 29194.878} C_VEL
LIN {X 0,Y 84.797,Z 748.275,A -85,B 0,C 180,E1 29195.256,E2 29195.256} C_VEL
LIN {X 0,Y 84.797,Z 862.5,A -85,B 0,C 180,E1 29195.256,E2 29195.256} C_VEL
LIN {X 0,Y 84.797,Z 862.5,A -85,B 0,C 180,E1 29195.256,E2 29195.256}

